	16#432D: sMsg := '432D parameter "Stepper motor stages for one speed stage not allowed" The value for the number of steps for each speed stage in the set value generation is not allowed.';
	16#432E: sMsg := '432E parameter "DWORD for the interpretation of the axis units not allowed" The value that contains the flags for the interpretation of the position and velocity units is not allowed.';
	16#432F: sMsg := '432F parameter "Maximum velocity not allowed" The value for the maximum permitted velocity is not allowed.';
	16#4330: sMsg := '4330 parameter "Motion monitoring window not allowed" The value for the motion monitoring window is not allowed. V';
	16#4331: sMsg := '4331 parameter "PEH time monitoring not allowed" The value for the activation of the PEH time monitoring is not allowed (PEH: positioning end and halt).';
	16#4332: sMsg := '4332 parameter "PEH monitoring time not allowed" The value for the PEH monitoring time (timeout) is not allowed (PEH: positioning end and halt). Default value: 5 s';
	16#4333: sMsg := '4333 parameter "AXISERR_RANGE_DELAYBREAKRELEASE"';
	16#4334: sMsg := '4334 parameter „AXISERR_RANGE_DATAPERSISTENCE”';
	16#433A: sMsg := '433A parameter „AXISERR_RANGE_POSDIFF_FADING_ACCELERATION”';
	16#433B: sMsg := '433B parameter "Fast Axis Stop Signal TYPE NOT allowed" The value FOR the Signal TYPE OF the Fast Axis StoP is NOT allowed [0...5].';
	16#4340: sMsg := '4340 initialization "Axis initialisation" Axis has not been initialised. Although the axis has been created, the rest of the initialisation has not been performed (1. Initialisation of axis I/O, 2. Initialisation of axis…';
	16#4341: sMsg := '4341 address "Group address" Axis does not have a group, or the group address has not been initialised (group contains the set value generation).';
	16#4342: sMsg := '4342 address "Encoder address" The axis does not have an encoder, or the encoder address has not been initialised.';
	16#4343: sMsg := '4343 address "Controller address" The axis does not have a controller, or the controller address has not been initialised.';
	16#4344: sMsg := '4344 address "Drive address" The axis does not have a drive, or the drive address has not been initialised.';
	16#4345: sMsg := '4345 address "Axis interface PLC to NC address" Axis does not have an axis interface from the PLC to the NC, or the axis interface address has not been initialised.';
	16#4346: sMsg := '4346 address "Axis interface NC to PLC address" Axis does not have an axis interface from the NC to the PLC, or the axis interface address has not been initialised.';
	16#4347: sMsg := '4347 address "Size of axis interface NC to PLC is not allowed" (INTERNAL ERROR) The size of the axis interface from NC to PLC is not allowed.';
	16#4348: sMsg := '4348 address "Size of axis interface PLC to NC is not allowed" (INTERNAL ERROR) The size of the axis interface from PLC to NC is not allowed.';
	16#4356: sMsg := '4356 monitoring "Controller enable" Controller enable for the axis is not present (see axis interface SPS®NC). This enable is required, for instance, for an axis positioning task.';
	16#4357: sMsg := '4357 monitoring "Feed enable minus" Feed enable for movement in the negative direction is not present (see axis interface SPS®NC). This enable is required, for instance, for an axis positioning task in the negative d…';
	16#4358: sMsg := '4358 monitoring "Feed enable plus" Feed enable for movement in the positive direction is not present (see axis interface SPS®NC). This enable is required, for instance, for an axis positioning task in the positive di…';
	16#4359: sMsg := '4359 monitoring "Set velocity not allowed" The set velocity requested for a positioning task is not allowed. This can happen if the velocity is less than or equal to zero, larger than the maximum permitted axis veloc…';
	16#435A: sMsg := '435A monitoring "Movement smaller than one encoder increment" (INTERNAL ERROR) The movement required of an axis is, in relation to a positioning task, smaller than one encoder increment (see scaling factor). This inf…';
	16#435B: sMsg := '435B monitoring "Set acceleration monitoring" (INTERNAL ERROR) The set acceleration has exceeded the maximum permitted acceleration or deceleration parameters of the axis.';
	16#435C: sMsg := '435C monitoring "PEH time monitoring" The PEH time monitoring has detected that, after the PEH monitoring time that follows a positioning has elapsed, the target position window has not been reached. The following po…';
	16#435D: sMsg := '435D monitoring "Encoder existence monitoring / movement monitoring" During the active positioning the actual encoder value has changed continuously for a default check time from NC cycle to NC cycle less than the de…';
	16#435E: sMsg := '435E monitoring „Looping distance less than breaking distance” The absolute value of the looping distance is less or equal than the positive or negative breaking distance. This is not allowed.';
	16#4361: sMsg := '4361 monitoring „Time range exceeded (future)” The calculated position lies too far in the future (e.g. when converting a position value in a DC time stamp).';
	16#4362: sMsg := '4362 monitoring „Time range exceeded (past)” The calculated position lies too far in the past (e.g. when converting a position value in a DC time stamp).';
	16#4363: sMsg := '4363 monitoring „Position cannot be determined” The requested position cannot be determined.';
	16#43A0: sMsg := '43A0 internal "Axis consequential error" Consequential error resulting from another causative error related to another axis. Axis consequential errors can occur in relation to master/slave couplings or with multipl…';
	16#4400: sMsg := '4400 parameter "Encoder ID not allowed" The value for the encoder ID is not allowed, e.g. because it has already been assigned, is less than or equal to zero, or is bigger than 255.';
	16#4401: sMsg := '4401 parameter "Encoder type not allowed" The value for the encoder type is unacceptable because it is not defined. Type 1: Simulation (incremental) Type 2: M3000 (24 bit absolute) Type 3: M31x0 (24 bit incremental)…';
	16#4402: sMsg := '4402 parameter "Encoder mode" The value for the encoder (operating) mode is not allowed. Mode 1: Determination of the actual position Mode 2: Determination of the actual position and the actual velocity (filter)';
	16#4403: sMsg := '4403 parameter "Encoder counting direction inverted?" The flag for the encoder counting direction is not allowed. Flag 0: Positive encoder counting direction Flag 1: Negative encoder counting direction';
	16#4404: sMsg := '4404 initialization "Referencing status" The flag for the referencing status is not allowed. Flag 0: Axis has not been referenced Flag 1: Axis has been referenced';
	16#4405: sMsg := '4405 parameter "Encoder increments for each physical encoder rotation" The value for the number of encoder increments for each physical rotation of the encoder is not allowed. This value is used by the software for …';
	16#4406: sMsg := '4406 parameter "Scaling factor" The value for the scaling factor is not allowed. This scaling factor provides the weighting for the conversion of an encoder increment (INC) to a physical unit such as millimeters or …';
	16#4407: sMsg := '4407 parameter "Position offset (zero point offset)" The value for the position offset of the encoder is not allowed. This value is added to the calculated encoder position, and is interpreted in the physical units …';
	16#4408: sMsg := '4408 parameter "Modulo factor" The value for the encoders modulo factor is not allowed.';
	16#4409: sMsg := '4409 parameter "Position filter time" The value for the actual position filter time is not allowed (P-T1 filter).';
	16#440A: sMsg := '440A parameter "Velocity filter time" The value for the actual velocity filter time is not allowed (P-T1 filter).';
	16#440B: sMsg := '440B parameter "Acceleration filter time" The value for the actual acceleration filter time is not allowed (P-T1 filter).';
	16#440C: sMsg := '440C initialization "Cycle time not allowed" (INTERNAL ERROR) The value of the SAF cycle time for the calculation of actual values is not allowed (e.g. is less than or equal to zero).';
	16#440D: sMsg := '440D initialization "" ENCERR_RANGE_UNITFLAGS';
	16#440E: sMsg := '440E parameter "Actual position correction / measurement system error correction" The value for the activation of the actual position correction ("measuring system error correction") is not allowed.';
	16#440F: sMsg := '440F parameter "Filter time actual position correction" The value for the actual position correction filter time is not allowed (P-T1 filter).';
	16#4410: sMsg := '4410 parameter "Search direction for referencing cam inverted" The value of the search direction of the referencing cam in a referencing procedure is not allowed. Value 0: Positive direction Value 1: Negative direct…';
	16#4411: sMsg := '4411 parameter "Search direction for sync pulse (zero pulse) inverted" The value of the search direction of the sync pulse (zero pulse) in a referencing procedure is not allowed. Value 0: Positive direction Value 1:…';
	16#4412: sMsg := '4412 parameter "Reference position" The value of the reference position in a referencing procedure is not allowed.';
	16#4413: sMsg := '4413 parameter "Clearance monitoring between activation of the hardware latch and appearance of the sync pulse" (NOT IMPLEMENTED) The flag for the clearance monitoring between activation of the hardware latch and oc…';
	16#4414: sMsg := '4414 parameter "Minimum clearance between activation of the hardware latch and appearance of the sync pulse" (NOT IMPLEMENTED) The value for the minimum clearance in increments between activation of the hardware lat…';
	16#4415: sMsg := '4415 parameter "External sync pulse" (NOT IMPLEMENTED) The value of the activation or deactivation of the external sync pulse in a referencing procedure is not allowed. Value 0: Passive Value 1: Active';
	16#4416: sMsg := '4416 parameter "Scaling of the noise rate is not allowed" The value of the scaling (weighting) of the synthetic noise rate is not allowed. This parameter exists only in the simulation encoder and serves to produce a…';
	16#4417: sMsg := '4417 parameter „Tolerance window for modulo-start” The value for the tolerance window for the modulo-axis-start is invalid. The value must be greater or equal than zero and smaller than the half encoder modulo-perio…';
	16#4418: sMsg := '4418 parameter „Encoder reference mode” The value for the encoder reference mode is not allowed, resp. is not supported for this encoder type.';
	16#4419: sMsg := '4419 parameter „Encoder evaluation direction” The value for the encoder evaluation direction (log. counter direction) is not allowed.';
	16#441A: sMsg := '441A parameter „Encoder reference system” The value for the encoder reference system is invalid (0: incremental, 1: absolute, 2: absolute+modulo).';
	16#441B: sMsg := '441B parameter „Encoder position initialization mode” When starting the TC system the value for the encoder position initialization mode is invalid.';
	16#441C: sMsg := '441C parameter „Encoder sign interpretation (UNSIGNED- / SIGNED- data type)” The value for the encoder sign interpretation (data type) for the encoder the actual increment calculation (0: Default/not defined, 1: UNS…';
	16#4420: sMsg := '4420 parameter "Software end location monitoring minimum not allowed" The value for the activation of the software location monitoring minimum is not allowed.';
	16#4421: sMsg := '4421 parameter "Software end location monitoring maximum not allowed" The value for the activation of the software location monitoring maximum is not allowed.';
	16#4422: sMsg := '4422 function "Actual value setting is outside the value range" The "set actual value" function cannot be carried out, because the new actual position is outside the expected range of values.';
	16#4423: sMsg := '4423 parameter "Software end location minimum not allowed" The value for the software end location minimum is not allowed.';
	16#4424: sMsg := '4424 parameter "Software end location maximum not allowed" The value for the software end location maximum is not allowed.';
	16#4425: sMsg := '4425 parameter „Filter mask for the raw data of the encoder is invalid” The value for the filter mask of the encoder raw data in increments is invalid.';
	16#4426: sMsg := '4426 parameter „Reference mask for the raw data of the encoder is invalid” The value for the reference mask (increments per encoder turn, absolute resolution) for the raw data of the encoder is invalid. E.g. this va…';
	16#4430: sMsg := '4430 function "Hardware latch activation (encoder)" Activation of the encoder hardware latch was implicitly initiated by the referencing procedure. If this function has already been activated but a latch value has …';
	16#4431: sMsg := '4431 function "External hardware latch activation (encoder)" The activation of the external hardware latch (only available on the KL5101) is initiated explicitly by an ADS command (called from the PLC program of th…';
	16#4432: sMsg := '4432 function "External hardware latch activation (encoder)" If a referencing procedure has previously been initiated and the hardware still signals a valid latch value ("latch valid"), this function must not be ca…';
	16#4433: sMsg := '4433 function "External hardware latch activation (encoder)" If this function has already been initiated and the hardware is still signaling that the external latch value is still valid ("extern latch valid"), a fu…';
	16#4434: sMsg := '4434 monitoring "Encoder function not supported" An encoder function has been activated that is currently not released for use, or which is not even implemented.';
	16#4435: sMsg := '4435 monitoring „Encoder function is already active” An encoder function can not been activated because this functionality is already active.';
	16#4440: sMsg := '4440 initialization "Encoder initialization" Encoder has not been initialized. Although the axis has been created, the rest of the initialization has not been performed (1. Initialization of axis I/O, 2. Initialization o…';
	16#4441: sMsg := '4441 address "Axis address" The encoder does not have an axis, or the axis address has not been initialized.';
	16#4442: sMsg := '4442 address "I/O input structure address" The drive does not have a valid I/O input address in the process image.';
	16#4443: sMsg := '4443 address "I/O output structure address" The encoder does not have a valid I/O output address in the process image.';
	16#4450: sMsg := '4450 monitoring "Encoder counter underflow monitoring" The encoders incremental counter has underflowed.';
	16#4451: sMsg := '4451 monitoring "Encoder counter overflow monitoring" The encoders incremental counter has overflowed.';
	16#4460: sMsg := '4460 monitoring "Software end location minimum (axis start)" With active monitoring of the software end location for a minimum, a start has been made from a position that lies below the software end location minimum.…';
	16#4461: sMsg := '4461 monitoring "Software end location maximum (axis start)" With active monitoring of the software end location for a maximum, a start has been made from a position that lies above the software end location maximum.…';
	16#4462: sMsg := '4462 monitoring "Software end location minimum (positioning process)" With active monitoring of the software end location for a minimum, the actual position has fallen below the software end location minimum. In the …';
	16#4463: sMsg := '4463 monitoring "Software end location maximum (positioning process)" With active monitoring of the software end location for a maximum, the actual position has exceeded the software end location maximum. In the case…';
	16#4464: sMsg := '4464 monitoring „Encoder hardware error” The drive resp. the encoder system reports a hardware error of the encoder. An optimal error code is displayed in the message of the event log.';
	16#4465: sMsg := '4465 monitoring „Position initialization error at system start” At the first initialization of the set position was this for all initialization trials (without over-/under-flow, with underflow and overflow ) out of t…';
	16#4470: sMsg := '4470 monitoring "SSI transformation fault or not finished" The SSI transformation of the FOX 50 module was faulty for some NC-cycles or did not finished respectively.';
	16#44A2: sMsg := '44A2 monitoring "ENCERR_ADDR_CONTROLLER"';
	16#44A3: sMsg := '44A3 monitoring "ENCERR_INVALID_CONTROLLERTYPE"';
	16#4500: sMsg := '4500 parameter "Controller ID not allowed" The value for the controller ID is not allowed, e.g. because it has already been assigned, is less than or equal to zero, or is greater than 255.';
	16#4501: sMsg := '4501 parameter "Controller type not allowed" The value for the controller type is unacceptable because it is not defined. Type 1: P-controller (position) . . . Type 7: High/low speed controller Type 8: Stepper motor…';
	16#4502: sMsg := '4502 parameter "Controller operating mode not allowed" The value for the controller operating mode is not allowed.';
	16#4503: sMsg := '4503 parameter "Weighting of the velocity pre-control not allowed" The value for the percentage weighting of the velocity pre-control is not allowed. The parameter is pre-set to 1.0 (100%) as standard.';
	16#4504: sMsg := '4504 parameter "Following error monitoring (position) not allowed" The value for the activation of the following error monitoring is not allowed.';
	16#4505: sMsg := '4505 parameter "Following error (velocity) not allowed" The value for the activation of the following error monitoring (velocity) is not allowed.';
	16#4506: sMsg := '4506 parameter "Following error window (position) not allowed" The value for the following error window (maximum allowable following error) is not allowed.';
	16#4507: sMsg := '4507 parameter "Following error filter time (position) not allowed" The value for the following error filter time (position) is not allowed.';
	16#4508: sMsg := '4508 parameter "Following error window (velocity) not allowed" The value for the following error window (velocity) is not allowed.';
	16#4509: sMsg := '4509 parameter "Following error filter time (velocity) not allowed" The value for the following error filter time (velocity) is not allowed.';
	16#4510: sMsg := '4510 parameter "Proportional gain Kv or Kp (position controller) not allowed" The value for the proportional gain (Kv factor or Kp factor) is not allowed.';
	16#4511: sMsg := '4511 parameter "Integral-action time Tn (position controller) not allowed" The value for the integral-action time is not allowed (I proportion of the PID T1 controller).';
	16#4512: sMsg := '4512 parameter "Derivative action time Tv (position controller) not allowed" The value for the derivative action time is not allowed (D proportion of the PID T1 controller).';
	16#4513: sMsg := '4513 parameter "Damping time Td (position controller) not allowed" The value for the damping time is not allowed (D proportion of the PID T1 controller). Suggested value: 0.1 * Tv';
	16#4514: sMsg := '4514 function "Activation of the automatic offset compensation not allowed" Activation of the automatic offset compensation is only possible for certain types of controller (with no I component).';
	16#4515: sMsg := '4515 parameter "Additional proportional gain Kv or Kp (position controller) not allowed" The value for the second term of the proportional gain (Kv factor or Kp factor) is not allowed.';
	16#4516: sMsg := '4516 parameter "Reference velocity for additional proportional gain Kv or Kp (position controller) not allowed" The value for the reference velocity percentage data entry, to which the additional proportional gain i…';
	16#4517: sMsg := '4517 parameter "Proportional gain Pa (acceleration proportion) not allowed" The value for the proportional gain (Pa factor) is not allowed.';
	16#4518: sMsg := '4518 parameter "Proportional gain Kv (velocity controller) not allowed" The value for the proportional gain (Kv factor) is not allowed.';
	16#4519: sMsg := '4519 parameter “Reset time Tn (velocity controller) not allowed” The value for the integral-action time is not allowed (I proportion of the PID T1 controller).';
	16#451A: sMsg := '451A address "CONTROLERR_RANGE_ACCJUMPLIMITINGMODE"';
	16#451B: sMsg := '451B address "CONTROLERR_RANGE_ACCJUMPVALUE"';
	16#451C: sMsg := '451C address "CONTROLERR_RANGE_FILTERTIME"';
	16#451D: sMsg := '451D parameter „Dead zone not allowed” The value for the dead zone from the position error or the velocity error (system deviation) is not allowed (only for complex controller with velocity or torque interface).';
	16#4520: sMsg := '4520 parameter ”Rate time Tv (velocity controller) not allowed” The value for the derivative action time is not allowed (D proportion of the PID T1 controller).';
	16#4521: sMsg := '4521 parameter "Damping time Td (velocity controller) not allowed" The value for the damping time is not allowed (D proportion of the PID T1 controller). Suggested value: 0.1 * Tv';
	16#4522: sMsg := '4522 parameter "CONTROLERR_RANGE_IOUTPUTLIMIT"';
	16#4523: sMsg := '4523 parameter "CONTROLERR_RANGE_DOUTPUTLIMIT"';
	16#4524: sMsg := '4524 parameter "CONTROLERR_RANGE_POSIDISABLEWHENMOVING"';
	16#4540: sMsg := '4540 initialization "Controller initialisation" Controller has not been initialised. Although the controller has been created, the rest of the initialisation has not been performed (1. Initialisation of controller, 2. Re…';
	16#4541: sMsg := '4541 address "Axis address" Controller does not know its axis, or the axis address has not been initialised.';
	16#4542: sMsg := '4542 address "Drive address" Controller does not know its drive, or the drive address has not been initialised.';
	16#4550: sMsg := '4550 monitoring "Following error monitoring (position)" With active following error monitoring (position) a following error exceedance has occurred, whose magnitude is greater than the following error window, and who…';
	16#4551: sMsg := '4551 monitoring "Following error monitoring (velocity)" With active following error monitoring (velocity) a velocity following error exceedance has occurred, whose magnitude is greater than the following error window…';
	16#45A0: sMsg := '45A0 monitoring "CONTROLERR_RANGE_AREA_ASIDE"';
	16#45A1: sMsg := '45A1 monitoring "CONTROLERR_RANGE_AREA_BSIDE"';
	16#45A2: sMsg := '45A2 monitoring "CONTROLERR_RANGE_QNENN"';
	16#45A3: sMsg := '45A3 monitoring "CONTROLERR_RANGE_PNENN"';
	16#45A4: sMsg := '45A4 monitoring "CONTROLERR_RANGE_AXISIDPRESP0"';
	16#4600: sMsg := '4600 parameter "Drive ID not allowed" The value for the drive ID is not allowed, e.g. because it has already been assigned, is less than or equal to zero, or is greater than 255.';
	16#4601: sMsg := '4601 parameter "Drive type not allowed" The value for the drive type is unacceptable because it is not defined.';
	16#4602: sMsg := '4602 parameter "Drive operating mode not allowed" The value for the drive operating mode is not allowed. Modus 1: Standard';
	16#4603: sMsg := '4603 parameter "Motor polarity inverted?" The flag for the motor polarity is not allowed. Flag 0: Positive motor polarity Flag 1: Negative motor polarity';
	16#4604: sMsg := '4604 parameter "Drift compensation/velocity offset (DAC offset)" The value for the drift compensation (DAC offset) is not allowed.';
	16#4605: sMsg := '4605 parameter "Reference velocity (velocity pre-control)" The value for the reference velocity (velocity pre-control) is not allowed.';
	16#4606: sMsg := '4606 parameter "Reference output in percent" The value for the reference output in percent is not allowed. The value 1.0 (100 %) usually corresponds to a voltage of 10.0 V.';
	16#4607: sMsg := '4607 parameter "Quadrant compensation factor" The value for the quadrant compensation factor is not allowed.';
	16#4608: sMsg := '4608 parameter "Velocity reference point in percent" The value for the velocity reference point in percent is not allowed. The value 1.0 corresponds to 100 percent.';
	16#4609: sMsg := '4609 parameter "Output reference point in percent" The value for the output reference point in percent is not allowed. The value 1.0 corresponds to 100 percent.';
	16#460A: sMsg := '460A parameter "Minimum or maximum output limit" The values for the minimum and/or maximum output limit is not allowed. This will happen if the range of values is exceeded, the maximum limit is smaller than the mini…';
	16#460B: sMsg := '460B parameter "DRIVEERR_RANGE_MAXINCREMENT"';
	16#460C: sMsg := '460C parameter "DRIVEERR_RANGE_ DRIVECONTROLDWORD"';
	16#460D: sMsg := '460D parameter "DRIVEERR_RANGE_ RESETCYCLECOUNTER"';
	16#460F: sMsg := '460F parameter „Drive torque output scaling is not allowed” The value for the drive torque output scaling (rotary motor) or the force output scaling (linear motor) is not allowed.';
	16#4610: sMsg := '4610 parameter „Drive velocity output scaling is not allowed” The value for the drive velocity output scaling is not allowed.';
	16#4611: sMsg := '4611 parameter "Profi Drive DSC Proportional gain Kpc (position controller) not allowed" The value for the profi drive DSC proportional gain (Kpc factor) is not allowed.';
	16#4612: sMsg := '4612 parameter „Table-ID is invalid” The value for the table-ID is invalid.';
	16#4613: sMsg := '4613 parameter „Table interpolationtype is invalid” The value for the table interpolation-type is invalid.';
	16#4614: sMsg := '4614 parameter „Outputoffset in percent is invalid” The value for the output offset in percent (+/- 1.0) is invalid.';
	16#4615: sMsg := '4615 parameter „Profi Drive DSC scaling factor for calculating Xerr (position controller) is not allowed” The value as profi drive DSC scaling factor for calculating Xerr is invalid.';
	16#4616: sMsg := '4616 parameter „Drive acceleration output scaling is not allowed” The value for the drive acceleration/deceleration output scaling is not allowed.';
	16#4617: sMsg := '4617 parameter „Drive position output scaling is not allowed” The value for the drive position output scaling is not allowed.';
	16#4620: sMsg := '4620 parameter "Bit mask for stepper motor cycle not allowed" A value in the various stepper motor masks for the cycle concerned is not allowed.';
	16#4621: sMsg := '4621 parameter "Bit mask for stepper motor holding current not allowed" The value for the stepper motor holding mask is not allowed.';
	16#4630: sMsg := '4630 monitoring „Overtemperature” The drive resp. terminal detects an overtemperature alarm.';
	16#4631: sMsg := '4631 monitoring „Undervoltage” The drive resp. terminal detects an undervoltage (supply voltage to low).';
	16#4632: sMsg := '4632 monitoring „Wire breakage in phase A” The drive resp. terminal detects a wire breakage in phase A.';
	16#4633: sMsg := '4633 monitoring „Wire breakage in phase B” The drive resp. terminal detects a wire breakage in phase B.';
	16#4634: sMsg := '4634 monitoring „Overcurrent in phase A” The drive resp. terminal detects an overcurrent in phase A.';
	16#4635: sMsg := '4635 monitoring „Overcurrent in Phase B” The drive resp. terminal detects an overcurrent in phase B.';
	16#4636: sMsg := '4636 monitoring „Torque overload (stall situation)” The drive resp. terminal detects a torque overload (stall situation).';
	16#4640: sMsg := '4640 initialization "Drive initialisation" Drive has not been initialised. Although the drive has been created, the rest of the initialisation has not been performed (1. Initialisation of drive I/O, 2. Initialisation of …';
	16#4641: sMsg := '4641 address "Axis address" Drive does not know its axis, or the axis address has not been initialised.';
	16#4642: sMsg := '4642 address "I/O input structure address" The drive does not have a valid I/O input address in the process image.';
	16#4643: sMsg := '4643 address "I/O output structure address" The drive does not have a valid I/O output address in the process image.';
	16#4650: sMsg := '4650 monitoring "Drive not ready for operation" The drive is not ready for operation. The following are possible causes: - the drive is in failure state (hardware fault) - the drive is in the starting-up stage…';
	16#4651: sMsg := '4651 monitoring "Error in cyclic communication with the drive (life counter)"';
	16#4652: sMsg := '4652 monitoring "Not permitted to change the table ID while the axis is enabled"';
	16#4655: sMsg := '4655 monitoring "Invalid IO data for more than n consecutive nc cycles"';
	16#4A00: sMsg := '4A00 parameter "Table ID not allowed" The value for the table ID is not allowed, e.g. because it has already been assigned, is less than or equal to zero, or is greater than 255.';
	16#4A01: sMsg := '4A01 parameter "Table type not allowed" The value for the table type is unacceptable because it is not defined.';
	16#4A02: sMsg := '4A02 parameter "Number of lines in the table not allowed" The value of the number of lines in the table is not allowed, because, for example, it is smaller than two at linear interpolation and smaller than four at s…';
	16#4A03: sMsg := '4A03 parameter "Number of columns in the table is not allowed" The value of the number of columns in the table is not allowed, because, for example, it is less than or equal to zero (depends upon the type of table o…';
	16#4A04: sMsg := '4A04 parameter "Step size (position delta) not allowed" The value for the step size between two lines (position delta) is not allowed, because, for example, it is less than or equal to zero.';
	16#4A05: sMsg := '4A05 parameter "Period not allowed" The value for the period is not allowed, because, for example, it is less than or equal to zero.';
	16#4A06: sMsg := '4A06 parameter "Table is not monotonic" The value for the step size is not allowed, because, for example, it is less than or equal to zero.';
	16#4A07: sMsg := '4A07 initialization „Table sub type is not allowed” The value for the table sub type is not allowed or otherwise the table class (slave type) do not match up to the table main type.';
	16#4A08: sMsg := '4A08 initialization „Table interpolation type is not allowed” The value for the table interpolation type is allowed.';
	16#4A09: sMsg := '4A09 initialization "Incorrect table main type" The table main type is unknown or otherwise the table class (slave type) do not match up to the table main type.';
	16#4A10: sMsg := '4A10 initialization "Table initialisation" Table has not been initialised. Although the table has been created, the rest of the initialisation has not been performed. For instance, the number of lines or columns may be l…';
	16#4A11: sMsg := '4A11 initialization "Not enough memory" Table could not be created, since there is not enough memory.';
	16#4A12: sMsg := '4A12 function "Function not executed, function not available" The function has not been implemented, or cannot be executed, for the present type of table.';
	16#4A13: sMsg := '4A13 function "Line index not allowed" The start line index or the stop line index to be used for read or write access to the table is not allowed. For instance, the line index may be greater than the total number …';
	16#4A14: sMsg := '4A14 function "Column index not allowed" The start column index or the stop column index to be used for read or write access to the table in not allowed. For instance, the column index may be greater than the total…';
	16#4A15: sMsg := '4A15 function "Number of lines not allowed" The number of lines to be read from or written to the table is not allowed. The number of lines must be an integer multiple of the number of elements in a line (n * numbe…';
	16#4A16: sMsg := '4A16 function "Number of columns not allowed" The number of columns to be read from or written to the table is not allowed. The number of columns must be an integer multiple of the number of elements in a column (n…';
	16#4A17: sMsg := '4A17 function "Error in scaling or in range entry" The entries in the table header are inconsistent, e.g. the validity range is empty. If the error is generated during the run time it is a run time error and stops …';
	16#4A18: sMsg := '4A18 function "Multi table slave out of range" The slave master position is outside the table values for the master. The error is a run-time error, and stops the master/slave group.';
	16#4A19: sMsg := '4A19 function "Solo table underflow" The slave master position is outside the table values for the master. The master value of the equidistant table, to be processed linearly, lies under the first table value. The …';
	16#4A1A: sMsg := '4A1A function "Solo table overflow" The slave master position is outside the table values for the master. The master value of the equidistant table, to be processed linearly, lies above the first table value. The e…';
	16#4A1B: sMsg := '4A1B parameter "Incorrect execution mode" The cyclic execution mode can only be "true" or "false".';
	16#4A1C: sMsg := '4A1C parameter "Impermissible parameter" The Fifo parameter is not allowed.';
	16#4A1D: sMsg := '4A1D parameter "Fifo is empty" The Fifo of the external generator is empty. This can signify end of track or a run time error.';
	16#4A1E: sMsg := '4A1E parameter "Fifo is full" The Fifo of the external generator is full. It is the user‘s task to continue to attempt to fill the Fifo with the rejected values.';
	16#4A1F: sMsg := '4A1F parameter „Point-Index of Motion Function invalid” The point index of a Motion Function Point of a Function Table is invalid. First the point index has to be larger than zero and second it has to be numerical c…';
	16#4A20: sMsg := '4A20 initialization „No diagonalisation of matrix” The spline can not be calculated. The master positions are not correct.';
	16#4A21: sMsg := '4A21 initialization „Number of spline points to less” The number of points of a cubic spline has to be greater than two.';
	16#4A22: sMsg := '4A22 initialization „Fifo must not be overwritten” Fifo must not be overwritten since then the active line would be overwritten. It is the task of the user to secure that the active line is not modified.';
	16#4B00: sMsg := '4B00 parameter "Axis has been stopped" The axis has been stopped while the axis moves to target position. The axis could be stopped with a PLC Command via ADS, with the call of AXFNC or with the TwinCAT System Manag…';
	16#4B01: sMsg := '4B01 parameter "Axis cannot be started" The axis cannot be started, because:';
	16#4B02: sMsg := '4B02 parameter "Control mode not allowed" No Target Position Control and no Position Area Control.';
	16#4B03: sMsg := '4B03 parameter "Axis is not moving" Restart position and velocity is only allowed if axis is physically moving.';
	16#4B04: sMsg := '4B04 parameter "Wrong mode for RestartPosAndVelo" Wrong mode.';
	16#4B05: sMsg := '4B05 parameter "Command not allowed"';
	16#4B06: sMsg := '4B06 parameter "Parameter not correct"';
	16#4B07: sMsg := '4B07 parameter "Timeout axis function block"';
	16#4B08: sMsg := '4B08 parameter "Axis in protected mode" Axis is in protected mode (i.e. coupled) and cannot be moved.';
	16#4B09: sMsg := '4B09 parameter "Axis is not ready" Axis is not ready and cannot be moved.';
	16#4B0A: sMsg := '4B0A parameter "Homing error" The Homing of an axis could not be started or was not successful';
	16#4B0B: sMsg := '4B0B parameter "Invalid definition trigger input definition" The definition of the trigger signal used with the function block MC_TouchProbe is invalid. The defined encoder ID, the trigger signal or the trigger sign…';
	16#4B0C: sMsg := '4B0C function "position latch has been deactivated" The function block MC_TouchProbe encountered that a touch probe sequence has been deactivated after the block started this sequence. The reason for instance can b…';
	16#4B0D: sMsg := '4B0D function "Timeout NC status feedback" A function block has successfully executed a command but the NC does not pass the expected feedback in the axis status word.';
	16#4B0E: sMsg := '4B0E function "Supplement not installed" - The function is available as supplement product but not installed on the system.';
	16#4B0F: sMsg := '4B0F function "Timeout Register Access" - The access to a bus terminal register timed out.';
	16#4B10: sMsg := '4B10 function "M-Function request missing" This error occurs if a confirmation of an M-Function is made but the request bit is not set.';
	16#4B11: sMsg := '4B11 parameter "Zero shift index is out of range" The index of the zero shift is invalid';
	16#4B12: sMsg := '4B12 parameter "R parameter index or size is invalid". This error occurs, if the R parameters are written or read and the index or size is out of range';
	16#4B13: sMsg := '4B13 parameter "Index for tool description is invalid"';
	16#4B14: sMsg := '4B14 function "Version of cyclic channel interface does not match to the requested function and function block, resp." This error occurs, if an older TwinCAT Version is used and a new functionality from a newer TcN…';
	16#4B15: sMsg := '4B15 function "Channel is not ready for requested function". The requested function can not be executed due to a wrong state of the channel. This error occurs for instance, if retrace is requested and the axes are …';
	16#4B16: sMsg := '4B16 function "Requested function is not turned on". The requested function requires an explicit activation before it can be executed.';
	16#4B20: sMsg := '4B20 parameter "Cannot append all axes". This error occurs, if you want to append an auxiliary axes to an interpolation group and the function fails. Probably a prior assignment of an auxiliary axes was skipped.';
	16#4B30: sMsg := '4B30 parameter "Pointer invalid". The pointer to a data structure is invalid, e.g. NULL.';
	16#4B31: sMsg := '4B31 parameter "Size of memory invalid". The size parameter is invalid.';
	16#4B32: sMsg := '4B32 parameter "Invalid cam table ID". The cam table ID is out of the range from 1 to 255.';
	16#4B33: sMsg := '4B33 parameter "Invalid point ID". The point ID of a motion function point is lower than 1.';
	16#4B34: sMsg := '4B34 parameter "Invalid number of points ". The number of points to read or write is less than 1.';
	16#4B35: sMsg := '4B35 parameter "Invalid MC table type". The type of a cam table does not match the MC_TableType definition.';
	16#4B36: sMsg := '4B36 parameter "Invalid number of rows". The number of rows of a cam table is less than 1.';
	16#4B37: sMsg := '4B37 parameter "Invalid number of columns". The number of columns of a cam table is invalid.';
	16#4B38: sMsg := '4B38 parameter "Invalid Increment". The increment for an interpolation is invalid, e.g. <= 0.';
	16#4B40: sMsg := '4B40 monitoring "Unsupported Terminal Type". The terminal in use is not supported by this function block.';
	16#4B41: sMsg := '4B41 monitoring "Register Read/Write Error". This error implies to be a validation error.';
	16#4B42: sMsg := '4B42 monitoring "Axis is Enabled". Axis is enabled and is not supposed to be enabled for this operation';
	16#4B43: sMsg := '4B43 parameter "Size of compensation table wrong". The stated table size in bytes is not conform with the real size.';
	16#4B44: sMsg := '4B44 parameter The minimum/ maximum position of the compenstation table is not conform to the position in the table description (ST_CompensationDesc)';
	16#4B45: sMsg := '4B45 parameter "Not implemented". The requested function is not implemented in this combination.';
	16#4B60: sMsg := '4B60 monitoring "Motion command not be activated". A motion command has been started and has been buffered and confirmed by the NC. Nevertheless the command did not become active.';
	16#4B61: sMsg := '4B61 monitoring "Motion command could not be monitored by the PLC". A motion command has been started and has been buffered and confirmed by the NC. The PLC has not been able to monitor the execution of this command……';
	16#4B62: sMsg := '4B62 monitoring "Buffered command finished with error". A buffered command finished with an error. The error number is not available because a new command is already in execution.';
	16#4B63: sMsg := '4B63 monitoring "Buffered command finished without state feedback". A buffered command finished without success or error feedback.';
	16#4B64: sMsg := '4B64 monitoring "  BufferMode  not supported". The  BufferMode  is not supported by the command.';
	16#4B65: sMsg := '4B65 monitoring "Command number is zero". The system administrated command number for buffered commands is zero. ';
	16#4B71: sMsg := '4B71 parameter "Invalid NCI Entry Type". FB_NciFeedTablePreparation is called with an unknown nEntryType';
	16#4B72: sMsg := '4B72 function "NciFeedTable full". The table is full filled and therefore this entry is not accepted.';
	16#4B73: sMsg := '4B73 function internal error';
	16#4B74: sMsg := '4B74 parameter "ST_NciTangentialFollowingDesc: tangential axis is not an auxiliary axis" The entry ST_NciTangentialFollowingDesc contains an tangential axis that is no auxiliary axis.';
	16#4B75: sMsg := '4B75 parameter ST_NciTangentialFollowingDesc: nPathAxis1 and nPathAxis2, resp. are no path axes. So it is not possible to determine the plane.';
	16#4B76: sMsg := '4B76 parameter ST_NciTangentialFollwoingDesc: nPathAxis1 and nPathAxis2 are equal. So it is not possible to determine the plane.';
	16#4B77: sMsg := '4B77 parameter ST_NciGeoCirclePlane: circle is programmed in a wrong manner.';
	16#4B78: sMsg := '4B78 function Internal error in calculation of the tangential following';
	16#4B79: sMsg := '4B79 monitoring Tangential following: With ST_NciTangentialFollowingDesc the monitoring of the deviation angle (E_TfErrorOnCrirical1) is activated and with the actual segment the deviation angle is too big.';
	16#4B7A: sMsg := '4B7A function not implemented';
	16#4B7B: sMsg := '4B7B parameter Tangential Following: The radius of the actual circle segment is too small';
	16#4B7C: sMsg := '4B7C parameter FB_NciFeedTablePreparation: pEntry is NULL';
	16#4B7D: sMsg := '4B7D parameter FB_NciFeedTablePreparation: The specified nEntryType does not match the the structure type';
	16#4B7E: sMsg := '4B7E parameter ST_NciMFuncFast and ST_NciMFuncHsk: The requested m-function is not in between 0..159';
	16#4B7F: sMsg := '4B7F parameter ST_NciDynOvr: The requested value for the dynamic override is not in between 0.01 and 1.0';
	16#4B80: sMsg := '4B80 parameter ST_NciVertexSmoothing: invalid parameter. This error occurs with a negative vertex radius or an unknown vertex smoothing type.';
	16#4B81: sMsg := '4B81 parameter FB_NciFeedTablePrepartion: The requested velocity is not in a valid range';
	16#4B82: sMsg := '4B82 parameter ST_Nci*: invalid parameter';

ELSE
	sMsg := UDINT_TO_STRING(iErrID);
	sMsg := concat(sMsg, ' Unknown Error code');
END_CASE
F_AxErrMsg := sMsg;

END_FUNCTION

// ---- POUs/POUsAxisOnline/AX5000/F_AX5xErrMsg.TcPOU
//==================================================================================================
//							Beckhoff Automation Poland
//								7.12.2018
//		Funkcja konwertujaca nr bledu na opis
// 	v1.0	|| TC v 3.1.4022.27	|| - pierwsza wersja
//==================================================================================================
FUNCTION F_AX5xErrMsg : STRING(255)
VAR_INPUT
	uiDriveError : UINT;
END_VAR

IF uiDriveError < 1 THEN
	F_AX5xErrMsg := '';
	RETURN;
END_IF

CASE uiDriveError OF
	16#1001: F_AX5xErrMsg:= '1001 =  No valid IDN';
	16#1009: F_AX5xErrMsg:= '1009 =  Invalid access to element 1';
	16#2001: F_AX5xErrMsg:= '2001 =  No name';
	16#2002: F_AX5xErrMsg:= '2002 =  Name transmission too short';
	16#2003: F_AX5xErrMsg:= '2003 =  Name transmission too long';
	16#2004: F_AX5xErrMsg:= '2004 =  Name cannot be changed';
	16#2005: F_AX5xErrMsg:= '2005 =  Name is write protected at this time';
	16#3002: F_AX5xErrMsg:= '3002 =  Attribute transmission too short';
	16#3003: F_AX5xErrMsg:= '3003 =  Attribute transmission too long';
	16#3004: F_AX5xErrMsg:= '3004 =  Attribute cannot be changed';
	16#3005: F_AX5xErrMsg:= '3005 =  Attribute is write protected at this time';
	16#4001: F_AX5xErrMsg:= '4001 =  No Unit';
	16#4002: F_AX5xErrMsg:= '4002 =  Unit transmission too short';
	16#4003: F_AX5xErrMsg:= '4003 =  Unit transmission too long';
	16#4004: F_AX5xErrMsg:= '4004 =  Unit cannot be changed';
	16#4005: F_AX5xErrMsg:= '4005 =  Unit is write protected at this time';
	16#5001: F_AX5xErrMsg:= '5001 =  No minimum input value';
	16#5002: F_AX5xErrMsg:= '5002 =  Minimum input value transmission too short';
	16#5003: F_AX5xErrMsg:= '5003 =  Minimum input value transmission too long';
	16#5004: F_AX5xErrMsg:= '5004 =  Minimum input value cannot be changed';
	16#5005: F_AX5xErrMsg:= '5005 =  Minimum input value is write protected at this time';
	16#6001: F_AX5xErrMsg:= '6001 =  No maximum input value';
	16#6002: F_AX5xErrMsg:= '6002 =  Maximum input value transmission too short';
	16#6003: F_AX5xErrMsg:= '6003 =  Maximum input value transmission too long';
	16#6004: F_AX5xErrMsg:= '6004 =  Maximum input value cannot be changed';
	16#6005: F_AX5xErrMsg:= '6005 =  Maximum input value is write protected at this time';
	16#7002: F_AX5xErrMsg:= '7002 =  Operation data value transmission too short';
	16#7003: F_AX5xErrMsg:= '7003 =  Operation data value transmission too long';
	16#7004: F_AX5xErrMsg:= '7004 =  Operation data value cannot be changed';
	16#7005: F_AX5xErrMsg:= '7005 =  Operation data value is write protected at this time';
	16#7006: F_AX5xErrMsg:= '7006 =  Operation data value is smaller than the minimum input value';
	16#7007: F_AX5xErrMsg:= '7007 =  Operation data value is greater than the maximum input value';
	16#7008: F_AX5xErrMsg:= '7008 =  Invalid operation data';
	16#7009: F_AX5xErrMsg:= '7009 =  Operation data is write protected by a password';
	16#7010: F_AX5xErrMsg:= '7010 =  Procedure command already active';
	16#7011: F_AX5xErrMsg:= '7011 =  Procedure command not interruptible';
	16#7012: F_AX5xErrMsg:= '7012 =  Procedure command is at this time not executable';
	16#7013: F_AX5xErrMsg:= '7013 =  Procedure command not executable';
	16#7014: F_AX5xErrMsg:= '7014 =  No data state';
	16#8001: F_AX5xErrMsg:= '8001 =  No default value';
	16#8002: F_AX5xErrMsg:= '8002 =  Default value transmission too long';
	16#8004: F_AX5xErrMsg:= '8004 =  Default value cannot be changed';
	16#700A: F_AX5xErrMsg:= '700A =  Operation data value is write protected';
	16#700B: F_AX5xErrMsg:= '700B =  Invalid indirect addressing';
	16#700C: F_AX5xErrMsg:= '700C =  Operation data is write protected due to other settings';
	16#700D: F_AX5xErrMsg:= '700D =  Reserved';
	16#800A: F_AX5xErrMsg:= '800A =  Invalid drive number';
	16#800B: F_AX5xErrMsg:= '800B =  General error';
	16#800C: F_AX5xErrMsg:= '800C =  No element addressed';
	16#CCD0: F_AX5xErrMsg:= 'CCD0 =  Leaving positive limit switch';
	16#CCD1: F_AX5xErrMsg:= 'CCD1 =  Leaving negative limit switch';
	16#CD40: F_AX5xErrMsg:= 'CD40 =  Clear warning: Overload internal brake resistor';
	16#CD41: F_AX5xErrMsg:= 'CD41 =  Clear warning: Overload external brake resistor';
	16#CD42: F_AX5xErrMsg:= 'CD42 =  Clear warning: Overtemperature amplifier';
	16#CD43: F_AX5xErrMsg:= 'CD43 =  Clear warning: Undervoltage DC link';
	16#CD46: F_AX5xErrMsg:= 'CD46 =  Clear warning: U_mains too high';
	16#CD47: F_AX5xErrMsg:= 'CD47 =  Clear warning: U_mains too low';
	16#D000: F_AX5xErrMsg:= 'D000 =  Esc state: Init';
	16#D001: F_AX5xErrMsg:= 'D001 =  Esc state: PreOp';
	16#D002: F_AX5xErrMsg:= 'D002 =  Esc state: Boot';
	16#D003: F_AX5xErrMsg:= 'D003 =  Esc state: SafeOp';
	16#D005: F_AX5xErrMsg:= 'D005 =  Esc state: Op';
	16#D006: F_AX5xErrMsg:= 'D006 =  Esc state: invalid';
	16#D010: F_AX5xErrMsg:= 'D010 =  Axis state machine: Control section not ready';
	16#D011: F_AX5xErrMsg:= 'D011 =  Axis state machine: Control section ready';
	16#D012: F_AX5xErrMsg:= 'D012 =  Axis state machine: Control and power section ready';
	16#D013: F_AX5xErrMsg:= 'D013 =  Axis state machine: Axis in operation';
	16#D014: F_AX5xErrMsg:= 'D014 =  Axis state machine: Axis halt';
	16#D015: F_AX5xErrMsg:= 'D015 =  Axis state machine: Axis error';
	16#D019: F_AX5xErrMsg:= 'D019 =  Axis state machine: Invalid state';
	16#D101: F_AX5xErrMsg:= 'D101 =  Hardware enable not active.';
	16#D102: F_AX5xErrMsg:= 'D102 =  Safety card active,  AX5000 in the safe condition';
	16#D180: F_AX5xErrMsg:= 'D180 =  SCI communication Control - Front pcb: Frame error';
	16#D181: F_AX5xErrMsg:= 'D181 =  SCI communication Control - Front pcb: Parity error';
	16#D182: F_AX5xErrMsg:= 'D182 =  SCI communication Control - Front pcb: RX-Data missing';
	16#D183: F_AX5xErrMsg:= 'D183 =  SCI communication Control - Front pcb: SCI error';
	16#D184: F_AX5xErrMsg:= 'D184 =  SCI communication Control - Front pcb: Timeout error';
	16#D185: F_AX5xErrMsg:= 'D185 =  SCI communication Control - Front pcb: Checksum error';
	16#D186: F_AX5xErrMsg:= 'D186 =  SCI communication Control - Front pcb: Byte count error';
	16#D187: F_AX5xErrMsg:= 'D187 =  SCI communication Control - Front pcb: Command denied';
	16#D188: F_AX5xErrMsg:= 'D188 =  SCI communication Control - Front pcb: Wrong command';
	16#D189: F_AX5xErrMsg:= 'D189 =  SCI communication Control - Front pcb: Command error';
	16#D18A: F_AX5xErrMsg:= 'D18A =  SCI communication Control - Front pcb: Timeout error';
	16#D18B: F_AX5xErrMsg:= 'D18B =  SCI communication Control - Front pcb: RX data error';
	16#D18C: F_AX5xErrMsg:= 'D18C =  SCI communication Control - Front pcb: Wrong channel';
	16#D18D: F_AX5xErrMsg:= 'D18D =  SCI communication Control - Front pcb: Fifo overflow';
	16#D18E: F_AX5xErrMsg:= 'D18E =  SCI communication Front - Control pcb: Frame error';
	16#D18F: F_AX5xErrMsg:= 'D18F =  SCI communication Front - Control pcb: Parity error';
	16#D190: F_AX5xErrMsg:= 'D190 =  SCI communication Front - Control pcb: Wrong checksum';
	16#D191: F_AX5xErrMsg:= 'D191 =  SCI communication Front - Control pcb: Timeout error';
	16#D192: F_AX5xErrMsg:= 'D192 =  SCI communication Front - Control pcb: Response timeout error';
	16#D193: F_AX5xErrMsg:= 'D193 =  SCI communication Front - Control pcb: Fifo overflow';
	16#D194: F_AX5xErrMsg:= 'D194 =  SCI communication Control - Front pcb: SCI reset called';
	16#D195: F_AX5xErrMsg:= 'D195 =  SCI communication Control - Front pcb: Byte count error';
	16#D196: F_AX5xErrMsg:= 'D196 =  SCI communication Control - Front pcb: Buffer overflow';
	16#D1B0: F_AX5xErrMsg:= 'D1B0 =  SCI communication Control - Option card: Frame error';
	16#D1B1: F_AX5xErrMsg:= 'D1B1 =  SCI communication Control - Option card: Parity error';
	16#D1B2: F_AX5xErrMsg:= 'D1B2 =  SCI communication Control - Option card: RX-Data missing';
	16#D1B3: F_AX5xErrMsg:= 'D1B3 =  SCI communication Control - Option card: SCI error';
	16#D1B4: F_AX5xErrMsg:= 'D1B4 =  SCI communication Control - Option card: Timeout error';
	16#D1B5: F_AX5xErrMsg:= 'D1B5 =  SCI communication Control - Option card: Checksum error';
	16#D1B6: F_AX5xErrMsg:= 'D1B6 =  SCI communication Control - Option card: Byte count error';
	16#D1B7: F_AX5xErrMsg:= 'D1B7 =  SCI communication Control - Option card: Command denied';
	16#D1B8: F_AX5xErrMsg:= 'D1B8 =  SCI communication Control - Option card: Wrong command';
	16#D1B9: F_AX5xErrMsg:= 'D1B9 =  SCI communication Control - Option card: Command error';
	16#D1BA: F_AX5xErrMsg:= 'D1BA =  SCI communication Control - Option card: Timeout error';
	16#D1BB: F_AX5xErrMsg:= 'D1BB =  SCI communication Control - Option card: RX data error';
	16#D1BC: F_AX5xErrMsg:= 'D1BC =  SCI communication Control - Option card: Wrong channel';
	16#D1BD: F_AX5xErrMsg:= 'D1BD =  SCI communication Control - Option card: Fifo overflow';
	16#D1BE: F_AX5xErrMsg:= 'D1BE =  SCI communication Front - Control pcb: Frame error';
	16#D1BF: F_AX5xErrMsg:= 'D1BF =  SCI communication Front - Control pcb: Parity error';
	16#D1C0: F_AX5xErrMsg:= 'D1C0 =  SCI communication Front - Control pcb: Wrong checksum';
	16#D1C1: F_AX5xErrMsg:= 'D1C1 =  SCI communication Front - Control pcb: Timeout error';
	16#D1C2: F_AX5xErrMsg:= 'D1C2 =  SCI communication Front - Control pcb: Response timeout error';
	16#D1C3: F_AX5xErrMsg:= 'D1C3 =  SCI communication Front - Control pcb: Fifo overflow';
	16#D1C4: F_AX5xErrMsg:= 'D1C4 =  SCI communication Control - Option card: SCI reset called';
	16#D1C5: F_AX5xErrMsg:= 'D1C5 =  SCI communication Control - Option card: Byte count error';
	16#D1C6: F_AX5xErrMsg:= 'D1C6 =  SCI communication Control - Option card: Buffer overflow';
	16#D200: F_AX5xErrMsg:= 'D200 =  Firmware update successful!';
	16#D400: F_AX5xErrMsg:= 'D400 =  ESC: PLL timeout';
	16#D401: F_AX5xErrMsg:= 'D401 =  ESC: Io-Sync timeout';
	16#D402: F_AX5xErrMsg:= 'D402 =  Info procedure command: state change';
	16#D403: F_AX5xErrMsg:= 'D403 =  Esc state machine: State change active';
	16#D404: F_AX5xErrMsg:= 'D404 =  Esc state machine: Error flag not cleared';
	16#D500: F_AX5xErrMsg:= 'D500 =  External ADC: Uref invalid';
	16#D780: F_AX5xErrMsg:= 'D780 =  Feedback Parameter Channel Endat: Crc Error';
	16#D781: F_AX5xErrMsg:= 'D781 =  Feedback Parameter Channel Endat: Mode crc error';
	16#D782: F_AX5xErrMsg:= 'D782 =  Feedback Parameter Channel Endat: Timeout encoder response';
	16#D783: F_AX5xErrMsg:= 'D783 =  Feedback Parameter Channel Endat: Timeout encoder response';
	16#D784: F_AX5xErrMsg:= 'D784 =  Feedback Parameter Channel Endat: Wrong response';
	16#D786: F_AX5xErrMsg:= 'D786 =  Feedback Parameter Channel Endat: Encoder not ready';
	16#D787: F_AX5xErrMsg:= 'D787 =  Feedback Parameter Channel Endat: Formatting OEM memory';
	16#D808: F_AX5xErrMsg:= 'D808 =  Feedback Parameter Channel Hiperface: Wrong analog channel';
	16#DC30: F_AX5xErrMsg:= 'DC30 =  I2C communication: Save error ID 1';
	16#DC31: F_AX5xErrMsg:= 'DC31 =  I2C communication: Save error ID 2';
	16#DC32: F_AX5xErrMsg:= 'DC32 =  I2C communication: Save parameter';
	16#DC33: F_AX5xErrMsg:= 'DC33 =  I2C communication: Save operation time 1';
	16#DC34: F_AX5xErrMsg:= 'DC34 =  I2C communication: Save operation time 2';
	16#DC35: F_AX5xErrMsg:= 'DC35 =  I2C communication: Read';
	16#DC36: F_AX5xErrMsg:= 'DC36 =  I2C communication: Read';
	16#DC37: F_AX5xErrMsg:= 'DC37 =  I2C communication: Read';
	16#DC38: F_AX5xErrMsg:= 'DC38 =  I2C communication: Write';
	16#DC39: F_AX5xErrMsg:= 'DC39 =  I2C communication: Write';
	16#DC3A: F_AX5xErrMsg:= 'DC3A =  I2C communication: Different operation time';
	16#DC3B: F_AX5xErrMsg:= 'DC3B =  I2C communication: Job buffer full';
	16#DC3C: F_AX5xErrMsg:= 'DC3C =  I2C communication: No safety hardware';
	16#DC3D: F_AX5xErrMsg:= 'DC3D =  I2C communication: No option hardware';
	16#DC3E: F_AX5xErrMsg:= 'DC3E =  I2C communication: Device operation time overflow';
	16#DC3F: F_AX5xErrMsg:= 'DC3F =  I2C communication: Channel operation time overflow';
	16#DCB0: F_AX5xErrMsg:= 'DCB0 =  Lcd: Wrong Esc state';
	16#DCB1: F_AX5xErrMsg:= 'DCB1 =  Lcd: Wrong axis state';
	16#DCB2: F_AX5xErrMsg:= 'DCB2 =  Lcd: Unknown cyclic job';
	16#DCB3: F_AX5xErrMsg:= 'DCB3 =  Lcd: Unknown job';
	16#DCB4: F_AX5xErrMsg:= 'DCB4 =  Lcd: Unknown state';
	16#DCB5: F_AX5xErrMsg:= 'DCB5 =  Lcd: Unknown state';
	16#DCB6: F_AX5xErrMsg:= 'DCB6 =  Lcd: Unknown state';
	16#DCB7: F_AX5xErrMsg:= 'DCB7 =  Lcd: Unknown state';
	16#DCB8: F_AX5xErrMsg:= 'DCB8 =  Lcd: Unknown menue state';
	16#DCB9: F_AX5xErrMsg:= 'DCB9 =  Lcd: Interface error';
	16#DCBA: F_AX5xErrMsg:= 'DCBA =  Lcd: Invalid state';
	16#DCBB: F_AX5xErrMsg:= 'DCBB =  Lcd: Communication error';
	16#DD42: F_AX5xErrMsg:= 'DD42 =  Power management: DC link current in limit';
	16#DD80: F_AX5xErrMsg:= 'DD80 =  Control pcb: Main loop time exceeded';
	16#DD81: F_AX5xErrMsg:= 'DD81 =  Control pcb: End of stack reached';
	16#DD82: F_AX5xErrMsg:= 'DD82 =  Front pcb: Main loop time exceeded';
	16#DD83: F_AX5xErrMsg:= 'DD83 =  Front pcb: End of stack reached';
	16#DFFF: F_AX5xErrMsg:= 'DFFF =  Debug firmware,  replace "As soon as possible"!';
	16#E160: F_AX5xErrMsg:= 'E160 =  Process data mapping: Mapping code of IDN %s could not be copied.';
	16#E290: F_AX5xErrMsg:= 'E290 =  High-priority processes cannot be processed';
	16#E300: F_AX5xErrMsg:= 'E300 =  The IO-Watchdog has been disabled!!!! (User mode debugging!)';
	16#E581: F_AX5xErrMsg:= 'E581 =  External Periphery - Control card: Reading the ESC-eeprom failed';
	16#ECD0: F_AX5xErrMsg:= 'ECD0 =  Positive limit switch warning.';
	16#ECD1: F_AX5xErrMsg:= 'ECD1 =  Negative limit switch warning.';
	16#ED00: F_AX5xErrMsg:= 'ED00 =  Motor overtemperature';
	16#ED01: F_AX5xErrMsg:= 'ED01 =  Overload - motor';
	16#ED40: F_AX5xErrMsg:= 'ED40 =  Overload - Internal brake resistor';
	16#ED41: F_AX5xErrMsg:= 'ED41 =  Overload - External brake resistor';
	16#ED42: F_AX5xErrMsg:= 'ED42 =  Overtemperature - Amplifier';
	16#ED43: F_AX5xErrMsg:= 'ED43 =  Undervoltage - DC link';
	16#ED46: F_AX5xErrMsg:= 'ED46 =  U_mains too high';
	16#ED47: F_AX5xErrMsg:= 'ED47 =  U_mains too low';
	16#ED60: F_AX5xErrMsg:= 'ED60 =  Feedback - Warning bit set';
	16#F010: F_AX5xErrMsg:= 'F010 =  Firmware-Download: Flash error';
	16#F011: F_AX5xErrMsg:= 'F011 =  Firmware-Download: Flash error';
	16#F012: F_AX5xErrMsg:= 'F012 =  Firmware-Download: Flash error';
	16#F013: F_AX5xErrMsg:= 'F013 =  Firmware-Download: Flash error';
	16#F014: F_AX5xErrMsg:= 'F014 =  Firmware-Download: Flash error';
	16#F015: F_AX5xErrMsg:= 'F015 =  Firmware-Download: Flash error';
	16#F016: F_AX5xErrMsg:= 'F016 =  Firmware-Download: Flash error';
	16#F017: F_AX5xErrMsg:= 'F017 =  Firmware-Download: Flash error';
	16#F018: F_AX5xErrMsg:= 'F018 =  Firmware-Download: Flash error';
	16#F019: F_AX5xErrMsg:= 'F019 =  Firmware-Download: Flash error';
	16#F01A: F_AX5xErrMsg:= 'F01A =  Firmware-Download: Flash error';
	16#F01B: F_AX5xErrMsg:= 'F01B =  Firmware-Download: Flash error';
	16#F01C: F_AX5xErrMsg:= 'F01C =  Firmware-Download: Flash error';
	16#F01D: F_AX5xErrMsg:= 'F01D =  Firmware-Download: Flash error';
	16#F01E: F_AX5xErrMsg:= 'F01E =  Firmware-Download: Flash error';
	16#F030: F_AX5xErrMsg:= 'F030 =  Firmware-Download: Invalid file name';
	16#F032: F_AX5xErrMsg:= 'F032 =  Firmware download: Firmware file does not match the device';
	16#F033: F_AX5xErrMsg:= 'F033 =  Firmware-Download: Firmware-File is defective';
	16#F040: F_AX5xErrMsg:= 'F040 =  Firmware-Download: Firmware-File is defective';
	16#F041: F_AX5xErrMsg:= 'F041 =  Firmware-Download: Firmware-File is defective';
	16#F042: F_AX5xErrMsg:= 'F042 =  Firmware-Download: Firmware-File is defective';
	16#F043: F_AX5xErrMsg:= 'F043 =  Firmware-Download: Read of the hardware ID"s failed.';
	16#F044: F_AX5xErrMsg:= 'F044 =  Firmware-Download: Firmware-File is wrong or defective';
	16#F045: F_AX5xErrMsg:= 'F045 =  Firmware-Download: Firmware-File is defective';
	16#F046: F_AX5xErrMsg:= 'F046 =  Firmware-Download: Firmware-File is defective';
	16#F047: F_AX5xErrMsg:= 'F047 =  Firmware-Download: Firmware-File is defective';
	16#F048: F_AX5xErrMsg:= 'F048 =  Firmware-Download: Hardware is defective';
	16#F049: F_AX5xErrMsg:= 'F049 =  Firmware-Download: Hardware is defective';
	16#F04A: F_AX5xErrMsg:= 'F04A =  Firmware-Download: Hardware is defective';
	16#F04B: F_AX5xErrMsg:= 'F04B =  Firmware-Download: Firmware-File is defective';
	16#F04C: F_AX5xErrMsg:= 'F04C =  Firmware-Download: Firmware-File is defective';
	16#F04D: F_AX5xErrMsg:= 'F04D =  Firmware-Download: Firmware-File is defective';
	16#F04E: F_AX5xErrMsg:= 'F04E =  Firmware-Download: Firmware-File is defective';
	16#F04F: F_AX5xErrMsg:= 'F04F =  Firmware-Download: Wrong TwinCAT version';
	16#F050: F_AX5xErrMsg:= 'F050 =  Firmware-Download: Firmware-File is defective';
	16#F051: F_AX5xErrMsg:= 'F051 =  Firmware-Download: Firmware-File is defective';
	16#F052: F_AX5xErrMsg:= 'F052 =  Firmware-Download: Firmware-File is defective';
	16#F053: F_AX5xErrMsg:= 'F053 =  Firmware-Download: Firmware-File is defective';
	16#F054: F_AX5xErrMsg:= 'F054 =  Firmware-Download: Firmware-File is defective';
	16#F055: F_AX5xErrMsg:= 'F055 =  Firmware-Download: Firmware-File is defective';
	16#F056: F_AX5xErrMsg:= 'F056 =  Firmware-Download: Firmware-File is wrong or defective';
	16#F057: F_AX5xErrMsg:= 'F057 =  Firmware-Download: Firmware-File is defective';
	16#F058: F_AX5xErrMsg:= 'F058 =  Firmware-Download: Firmware-File is defective';
	16#F059: F_AX5xErrMsg:= 'F059 =  Firmware-Download: Firmware-File is defective';
	16#F060: F_AX5xErrMsg:= 'F060 =  Firmware-Download: Firmware-File is defective';
	16#F061: F_AX5xErrMsg:= 'F061 =  Firmware-Download: Hardware is defective';
	16#F062: F_AX5xErrMsg:= 'F062 =  Firmware-Download: Hardware is defective';
	16#F063: F_AX5xErrMsg:= 'F063 =  Firmware-Download: Firmware-File or device is defective';
	16#F064: F_AX5xErrMsg:= 'F064 =  Firmware-Download: Firmware-File or device is defective';
	16#F065: F_AX5xErrMsg:= 'F065 =  Firmware-Download: Firmware-File is wrong';
	16#F066: F_AX5xErrMsg:= 'F066 =  Firmware-Download: Firmware-File or device is defective';
	16#F067: F_AX5xErrMsg:= 'F067 =  Firmware-Download: Internal config error';
	16#F068: F_AX5xErrMsg:= 'F068 =  Firmware-Download: Bootloader update required.';
	16#F06A: F_AX5xErrMsg:= 'F06A =  Firmware-Download: Ctrl pcb eeprom not accessible.';
	16#F06B: F_AX5xErrMsg:= 'F06B =  Firmware-Download: Front pcb eeprom not accessible.';
	16#F06C: F_AX5xErrMsg:= 'F06C =  Firmware-Download: Driver pcb eeprom not accessible.';
	16#F06D: F_AX5xErrMsg:= 'F06D =  Firmware-Download: Power pcb eeprom not accessible.';
	16#F06E: F_AX5xErrMsg:= 'F06E =  Firmware-Download: Safety pcb eeprom not accessible.';
	16#F06F: F_AX5xErrMsg:= 'F06F =  Firmware-Download: Safety pcb eeprom not accessible.';
	16#F070: F_AX5xErrMsg:= 'F070 =  Firmware-Download: Firmware index for the control pcb don"t match';
	16#F071: F_AX5xErrMsg:= 'F071 =  Firmware-Download: Firmware index for the front pcb don"t match';
	16#F072: F_AX5xErrMsg:= 'F072 =  Firmware-Download: Firmware index for the driver pcb don"t match';
	16#F073: F_AX5xErrMsg:= 'F073 =  Firmware-Download: Firmware index for the power pcb don"t match';
	16#F074: F_AX5xErrMsg:= 'F074 =  Firmware-Download: Firmware index for the Safety pcb don"t match';
	16#F075: F_AX5xErrMsg:= 'F075 =  Firmware-Download: Firmware index for the option pcb don"t match';
	16#F076: F_AX5xErrMsg:= 'F076 =  Firmware-Download: Firmware index for the control pcb can"t be read';
	16#F077: F_AX5xErrMsg:= 'F077 =  Firmware-Download: Firmware index for the front pcb can"t be read';
	16#F078: F_AX5xErrMsg:= 'F078 =  Firmware-Download: Firmware index for the driver pcb can"t be read';
	16#F079: F_AX5xErrMsg:= 'F079 =  Firmware-Download: Firmware index for the power pcb can"t be read';
	16#F07A: F_AX5xErrMsg:= 'F07A =  Firmware-Download: Firmware index for the safety pcb can"t be read';
	16#F07B: F_AX5xErrMsg:= 'F07B =  Firmware-Download: Firmware index for the option pcb can"t be read';
	16#F090: F_AX5xErrMsg:= 'F090 =  Firmware-Download: FPGA error option pcb';
	16#F091: F_AX5xErrMsg:= 'F091 =  Firmware-Download: FPGA error option pcb';
	16#F092: F_AX5xErrMsg:= 'F092 =  Firmware-Download: FPGA error option pcb';
	16#F093: F_AX5xErrMsg:= 'F093 =  Firmware-Download: FPGA error option pcb';
	16#F094: F_AX5xErrMsg:= 'F094 =  Firmware-Download: FPGA error option pcb';
	16#F095: F_AX5xErrMsg:= 'F095 =  Firmware-Download: FPGA error option pcb';
	16#F096: F_AX5xErrMsg:= 'F096 =  Firmware-Download: FPGA error option pcb';
	16#F0A0: F_AX5xErrMsg:= 'F0A0 =  FPGA error: configuration could not be loaded';
	16#F0A1: F_AX5xErrMsg:= 'F0A1 =  FPGA error: Configuration file is missing';
	16#F0A2: F_AX5xErrMsg:= 'F0A2 =  FPGA error: Loading of the configuration failed.';
	16#F0B0: F_AX5xErrMsg:= 'F0B0 =  Serial Flash error';
	16#F0B1: F_AX5xErrMsg:= 'F0B1 =  Serial Flash error';
	16#F0B2: F_AX5xErrMsg:= 'F0B2 =  Serial Flash error';
	16#F0B3: F_AX5xErrMsg:= 'F0B3 =  Serial Flash error';
	16#F0B4: F_AX5xErrMsg:= 'F0B4 =  Serial Flash error';
	16#F0B5: F_AX5xErrMsg:= 'F0B5 =  Serial Flash error';
	16#F0B6: F_AX5xErrMsg:= 'F0B6 =  Serial Flash error';
	16#F0B7: F_AX5xErrMsg:= 'F0B7 =  Serial Flash error';
	16#F0B8: F_AX5xErrMsg:= 'F0B8 =  Serial Flash error';
	16#F0B9: F_AX5xErrMsg:= 'F0B9 =  Serial Flash error: Bootloader defective';
	16#F0BA: F_AX5xErrMsg:= 'F0BA =  Serial Flash error: Internal firmware file is defective';
	16#F0BB: F_AX5xErrMsg:= 'F0BB =  Serial Flash error: Internal system data file not found';
	16#F0BC: F_AX5xErrMsg:= 'F0BC =  Serial Flash error: Internal system data file is defective';
	16#F0BD: F_AX5xErrMsg:= 'F0BD =  Serial Flash error: Initialization failed';
	16#F0BE: F_AX5xErrMsg:= 'F0BE =  Serial Flash error: Processing failed';
	16#F0BF: F_AX5xErrMsg:= 'F0BF =  Serial Flash error: Write error';
	16#F0C0: F_AX5xErrMsg:= 'F0C0 =  Serial Flash error: Diagnostics file not found';
	16#F0C1: F_AX5xErrMsg:= 'F0C1 =  Serial Flash error: Internal error';
	16#F100: F_AX5xErrMsg:= 'F100 =  Axis state machine: Communication error';
	16#F101: F_AX5xErrMsg:= 'F101 =  Axis state machine: Initialize error';
	16#F102: F_AX5xErrMsg:= 'F102 =  Axis state machine: Loss of the hardware enable';
	16#F103: F_AX5xErrMsg:= 'F103 =  Axis state machine: Got no timer';
	16#F104: F_AX5xErrMsg:= 'F104 =  Axis state machine: NC errorhandling - Timeout';
	16#F105: F_AX5xErrMsg:= 'F105 =  Axis state machine: Maximum drive off delay time elapsed';
	16#F106: F_AX5xErrMsg:= 'F106 =  Axis state machine: No motor configured';
	16#F107: F_AX5xErrMsg:= 'F107 =  Axis state machine: Current control not ready to enable';
	16#F108: F_AX5xErrMsg:= 'F108 =  Axis state machine: Velocity control not ready';
	16#F109: F_AX5xErrMsg:= 'F109 =  Axis state machine: Position control not ready';
	16#F10A: F_AX5xErrMsg:= 'F10A =  Axis state machine: Wake and Shake not idle';
	16#F10B: F_AX5xErrMsg:= 'F10B =  Axis State Machine: Wake and Shake command failed';
	16#F10C: F_AX5xErrMsg:= 'F10C =  Axis State Machine: Not possible to enable';
	16#F10D: F_AX5xErrMsg:= 'F10D =  Axis State Machine: Not possible to enable';
	16#F10E: F_AX5xErrMsg:= 'F10E =  Axis State Machine: The motor connection check failed.';
	16#F10F: F_AX5xErrMsg:= 'F10F =  Axis State Machine: The configured error propagation input isn"t active.';
	16#F120: F_AX5xErrMsg:= 'F120 =  Command "Motor and feedback check": Timeout';
	16#F121: F_AX5xErrMsg:= 'F121 =  Command "Motor and feedback check": No hardware enable';
	16#F122: F_AX5xErrMsg:= 'F122 =  Command "Motor and feedback connection check"';
	16#F123: F_AX5xErrMsg:= 'F123 =  Command "Motor and feedback check" failed';
	16#F124: F_AX5xErrMsg:= 'F124 =  Reset-Command: Got no timer';
	16#F125: F_AX5xErrMsg:= 'F125 =  Reset-Command: Got no timer';
	16#F126: F_AX5xErrMsg:= 'F126 =  Reset-Command: Initialization failed';
	16#F127: F_AX5xErrMsg:= 'F127 =  Reset-Command: Feedback DSP - timeout';
	16#F128: F_AX5xErrMsg:= 'F128 =  Reset-Command: One or more of the pending errors is not resettable';
	16#F129: F_AX5xErrMsg:= 'F129 =  Reset-Command: Reset is not executable';
	16#F12A: F_AX5xErrMsg:= 'F12A =  Error reaction "Torque off" forced';
	16#F12B: F_AX5xErrMsg:= 'F12B =  Error reaction "Shorted coils brake" forced';
	16#F12C: F_AX5xErrMsg:= 'F12C =  Error reaction "Open loop ramp" forced';
	16#F12D: F_AX5xErrMsg:= 'F12D =  Error reaction "Closed loop ramp" forced';
	16#F12E: F_AX5xErrMsg:= 'F12E =  Error reaction "NC-Handling" forced';
	16#F12F: F_AX5xErrMsg:= 'F12F =  Command "Motor and feedback connection check": No enable permission from the Safety option';
	16#F130: F_AX5xErrMsg:= 'F130 =  Command "Wake and Shake": Timeout';
	16#F131: F_AX5xErrMsg:= 'F131 =  Command "Reset": Feedback initialization failed';
	16#F132: F_AX5xErrMsg:= 'F132 =  Command "Reset": Not possible - Internal hardware error';
	16#F133: F_AX5xErrMsg:= 'F133 =  Command "Reset": Not possible - Drive is still enabled';
	16#F134: F_AX5xErrMsg:= 'F134 =  Command "Reset": Restart of the modulo calculation failed.';
	16#F135: F_AX5xErrMsg:= 'F135 =  Parameterset-Switching: Reactivation of the parameterset 0 failed.';
	16#F136: F_AX5xErrMsg:= 'F136 =  Parameterset-Switching: Switching to parameterset x failed.';
	16#F137: F_AX5xErrMsg:= 'F137 =  Parameterset-Switching: Feature not available';
	16#F138: F_AX5xErrMsg:= 'F138 =  Parameterset-Switching: Axis is in operation,  switching not possible. ';
	16#F139: F_AX5xErrMsg:= 'F139 =  Parameterset-Switching: Internal error.';
	16#F13A: F_AX5xErrMsg:= 'F13A =  Parameterset-Switching: Switching to parameterset x not possible.';
	16#F13B: F_AX5xErrMsg:= 'F13B =  Option card and OCT interface: Reset failed.';
	16#F13C: F_AX5xErrMsg:= 'F13C =  Reset command - Timeout';
	16#F13E: F_AX5xErrMsg:= 'F13E =  error reaction ôFeedback errorö forced';
	16#F13F: F_AX5xErrMsg:= 'F13F =  Creation of the position interpolator failed';
	16#F140: F_AX5xErrMsg:= 'F140 =  Build drive system: Failed';
	16#F141: F_AX5xErrMsg:= 'F141 =  Build drive system: Timeout';
	16#F142: F_AX5xErrMsg:= 'F142 =  Initialization of the current controller failed';
	16#F143: F_AX5xErrMsg:= 'F143 =  Initialization of the velocity controller failed';
	16#F144: F_AX5xErrMsg:= 'F144 =  Initialization of the position controller failed';
	16#F145: F_AX5xErrMsg:= 'F145 =  Initialization of the feedback failed';
	16#F146: F_AX5xErrMsg:= 'F146 =  Build drive system: Failed';
	16#F147: F_AX5xErrMsg:= 'F147 =  Build drive system: Memory error Front card';
	16#F148: F_AX5xErrMsg:= 'F148 =  Build drive system: Unknown feedback system';
	16#F149: F_AX5xErrMsg:= 'F149 =  Build drive system: Front card - Internal error';
	16#F14A: F_AX5xErrMsg:= 'F14A =  Build drive system: Front card û software error';
	16#F14B: F_AX5xErrMsg:= 'F14B =  Build drive system: Memory error Control card';
	16#F14C: F_AX5xErrMsg:= 'F14C =  Build drive system: Memory error Front card';
	16#F14D: F_AX5xErrMsg:= 'F14D =  System memory deallocation: Feedback termination failed';
	16#F14E: F_AX5xErrMsg:= 'F14E =  System memory deallocation: Command error';
	16#F14F: F_AX5xErrMsg:= 'F14F =  System memory deallocation: Command error';
	16#F150: F_AX5xErrMsg:= 'F150 =  Initialization of the feedback: Internal error';
	16#F151: F_AX5xErrMsg:= 'F151 =  Initialization of the feedback: Timeout';
	16#F152: F_AX5xErrMsg:= 'F152 =  Initialisation of the feedback: Command failed';
	16#F153: F_AX5xErrMsg:= 'F153 =  Initialization of the feedback: No option card found';
	16#F154: F_AX5xErrMsg:= 'F154 =  Build drive system: Memory error option card';
	16#F155: F_AX5xErrMsg:= 'F155 =  Build drive system: Option card - Unknown feedback system';
	16#F156: F_AX5xErrMsg:= 'F156 =  Build drive system: Option card - Internal error';
	16#F157: F_AX5xErrMsg:= 'F157 =  Build drive system: Option card - Unknown feedback system';
	16#F158: F_AX5xErrMsg:= 'F158 =  System memory deallocation: Front card - Internal error';
	16#F159: F_AX5xErrMsg:= 'F159 =  System memory deallocation: Option card - Internal error';
	16#F15A: F_AX5xErrMsg:= 'F15A =  Feedback error: Plug connector combination invalid';
	16#F15B: F_AX5xErrMsg:= 'F15B =  Feedback error: No OCT support.';
	16#F15F: F_AX5xErrMsg:= 'F15F =  No control loops allocated. Calibration mode active.';
	16#F160: F_AX5xErrMsg:= 'F160 =  Process data mapping: Internal error';
	16#F161: F_AX5xErrMsg:= 'F161 =  Process data mapping: AT - S-0-0016';
	16#F162: F_AX5xErrMsg:= 'F162 =  Process data mapping: AT - S-0-0016';
	16#F163: F_AX5xErrMsg:= 'F163 =  Process data mapping: AT - Memory problem';
	16#F164: F_AX5xErrMsg:= 'F164 =  Process data mapping: Internal error';
	16#F165: F_AX5xErrMsg:= 'F165 =  Process data mapping: AT - Anzahl der IDN"s';
	16#F166: F_AX5xErrMsg:= 'F166 =  Process data mapping: MDT - S-0-0024';
	16#F167: F_AX5xErrMsg:= 'F167 =  Process data mapping: MDT - S-0-0024';
	16#F168: F_AX5xErrMsg:= 'F168 =  Process data mapping: MDT - Memory problem';
	16#F169: F_AX5xErrMsg:= 'F169 =  Process data mapping: Internal error';
	16#F16A: F_AX5xErrMsg:= 'F16A =  Process data mapping: MDT - Too many IDN"s';
	16#F16B: F_AX5xErrMsg:= 'F16B =  Process data mapping: AT-list,  double listed entry found';
	16#F16C: F_AX5xErrMsg:= 'F16C =  Process data mapping: MDT-list,  double listed entry found';
	16#F180: F_AX5xErrMsg:= 'F180 =  Internal communication: SCI - Control card to front card';
	16#F183: F_AX5xErrMsg:= 'F183 =  Feedback (general): Commutation feedback is not feedback 1';
	16#F184: F_AX5xErrMsg:= 'F184 =  Feedback "general": Commutation feedback is not feedback 2';
	16#F185: F_AX5xErrMsg:= 'F185 =  Internal communication: SCI - Control card to front card';
	16#F186: F_AX5xErrMsg:= 'F186 =  Internal communication: SCI - Control card to front card';
	16#F187: F_AX5xErrMsg:= 'F187 =  Internal communication: SCI - Control card to front card';
	16#F188: F_AX5xErrMsg:= 'F188 =  Internal communication: SCI - Control card to front card';
	16#F189: F_AX5xErrMsg:= 'F189 =  Internal communication: SCI - Control card to front card';
	16#F18A: F_AX5xErrMsg:= 'F18A =  Internal communication: SCI - Control card to front card';
	16#F18B: F_AX5xErrMsg:= 'F18B =  Internal communication: SCI - Control card to front card';
	16#F18C: F_AX5xErrMsg:= 'F18C =  Internal communication: SCI - Front card to control card';
	16#F18D: F_AX5xErrMsg:= 'F18D =  Internal communication: SCI - Front card to control card';
	16#F18E: F_AX5xErrMsg:= 'F18E =  Internal communication: SCI - Front card to control card';
	16#F18F: F_AX5xErrMsg:= 'F18F =  Internal communication: SCI - Front card to control card';
	16#F190: F_AX5xErrMsg:= 'F190 =  Internal communication: SPI - Control card to front card';
	16#F191: F_AX5xErrMsg:= 'F191 =  Internal communication: SPI - Control card to front card';
	16#F192: F_AX5xErrMsg:= 'F192 =  Internal communication: SPI - Control card to front card';
	16#F193: F_AX5xErrMsg:= 'F193 =  Internal communication: SPI - Control card to front card';
	16#F194: F_AX5xErrMsg:= 'F194 =  Internal communication: SPI - Front card to Control card';
	16#F195: F_AX5xErrMsg:= 'F195 =  Internal communication: SPI - Front card to Control card';
	16#F196: F_AX5xErrMsg:= 'F196 =  Internal communication: SPI - Front card to Control card';
	16#F197: F_AX5xErrMsg:= 'F197 =  Internal communication: SPI - Front card to Control card';
	16#F198: F_AX5xErrMsg:= 'F198 =  Internal communication: SPI - Control card to front card';
	16#F199: F_AX5xErrMsg:= 'F199 =  Internal communication: SPI - Control card to front card';
	16#F19A: F_AX5xErrMsg:= 'F19A =  Internal communication: SPI - Control card to front card';
	16#F19B: F_AX5xErrMsg:= 'F19B =  Internal communication: SPI - Control card to front card';
	16#F19C: F_AX5xErrMsg:= 'F19C =  Internal communication: SPI - Control card to front card';
	16#F19D: F_AX5xErrMsg:= 'F19D =  Internal communication: SPI - Control card to front card';
	16#F19E: F_AX5xErrMsg:= 'F19E =  Internal communication: SPI - Control card to front card';
	16#F1A0: F_AX5xErrMsg:= 'F1A0 =  Internal communication: SCI - Control card to front card';
	16#F1A1: F_AX5xErrMsg:= 'F1A1 =  Internal communication: SCI - Control card to front card';
	16#F1B0: F_AX5xErrMsg:= 'F1B0 =  Communication Control - Option pcb: Init failed.';
	16#F1B1: F_AX5xErrMsg:= 'F1B1 =  Option slot card: Commutation feedback not supported.';
	16#F1B2: F_AX5xErrMsg:= 'F1B2 =  Option slot card: Additional feedback not feedback 2.';
	16#F1B5: F_AX5xErrMsg:= 'F1B5 =  Internal communication: SCI - Control card to option card';
	16#F1B6: F_AX5xErrMsg:= 'F1B6 =  Internal communication: SCI - Control card to option card';
	16#F1B7: F_AX5xErrMsg:= 'F1B7 =  Internal communication: SCI - Control card to option card';
	16#F1B8: F_AX5xErrMsg:= 'F1B8 =  Internal communication: SCI - Control card to option card';
	16#F1B9: F_AX5xErrMsg:= 'F1B9 =  Internal communication: SCI - Control card to option card';
	16#F1BA: F_AX5xErrMsg:= 'F1BA =  Internal communication: SCI - Control card to option card';
	16#F1BB: F_AX5xErrMsg:= 'F1BB =  Internal communication: SCI - Control card to option card';
	16#F1BC: F_AX5xErrMsg:= 'F1BC =  Internal communication: SPI - Control card to option card';
	16#F1BD: F_AX5xErrMsg:= 'F1BD =  Internal communication: SPI - Control card to option card';
	16#F1D0: F_AX5xErrMsg:= 'F1D0 =  Internal communication: SCI - Control card to option card';
	16#F1D1: F_AX5xErrMsg:= 'F1D1 =  Internal communication: The feedback unit don"t supports the requested action.';
	16#F290: F_AX5xErrMsg:= 'F290 =  Cycle time out: High prioritise processes';
	16#F291: F_AX5xErrMsg:= 'F291 =  Time out: Low prioritise processes';
	16#F292: F_AX5xErrMsg:= 'F292 =  Internal task scheduler error';
	16#F2A0: F_AX5xErrMsg:= 'F2A0 =  Commutation error';
	16#F2A1: F_AX5xErrMsg:= 'F2A1 =  Overcurrent error motor, measuring limit reached (X13 / X23).';
	16#F2A2: F_AX5xErrMsg:= 'F2A2 =  Processing unit periphery: Initialisation failed';
	16#F2A3: F_AX5xErrMsg:= 'F2A3 =  Current controler: Internal use failed';
	16#F2A4: F_AX5xErrMsg:= 'F2A4 =  Internal error';
	16#F2A5: F_AX5xErrMsg:= 'F2A5 =  Internal error';
	16#F2A7: F_AX5xErrMsg:= 'F2A7 =  Torque off triggered from "shorted coils brake" or "DC brake"';
	16#F2E1: F_AX5xErrMsg:= 'F2E1 =  Velocity Control: Control deviation monitoring failed';
	16#F320: F_AX5xErrMsg:= 'F320 =  Discontinuity in the position command value';
	16#F321: F_AX5xErrMsg:= 'F321 =  Excessive position deviation';
	16#F323: F_AX5xErrMsg:= 'F323 =  Parameter error';
	16#F324: F_AX5xErrMsg:= 'F324 =  Excessive position command value deviation.';
	16#F325: F_AX5xErrMsg:= 'F325 =  Following distance calculation limit exceeded.';
	16#F326: F_AX5xErrMsg:= 'F326 =  Additional position deviation monitoring';
	16#F330: F_AX5xErrMsg:= 'F330 =  Position control - Interpolator error';
	16#F331: F_AX5xErrMsg:= 'F331 =  Position control - Interpolator error';
	16#F332: F_AX5xErrMsg:= 'F332 =  Position control - Interpolator error';
	16#F333: F_AX5xErrMsg:= 'F333 =  Position control - Interpolator error';
	16#F340: F_AX5xErrMsg:= 'F340 =  Position offset invalid';
	16#F341: F_AX5xErrMsg:= 'F341 =  Position offset: No position offset excisting';
	16#F342: F_AX5xErrMsg:= 'F342 =  Position offset: Offset can"t be activated. Modulo calculation is active.';
	16#F343: F_AX5xErrMsg:= 'F343 =  Position offset: No position offset excisting';
	16#F344: F_AX5xErrMsg:= 'F344 =  Position offset: The position offset change is greater than the modulo value.';
	16#F350: F_AX5xErrMsg:= 'F350 =  Modulo Calculation: No saved data could be loaded.';
	16#F351: F_AX5xErrMsg:= 'F351 =  Modulo Calculation: Initialization data invalid.';
	16#F352: F_AX5xErrMsg:= 'F352 =  Modulo Calculation: No saved data available.';
	16#F353: F_AX5xErrMsg:= 'F353 =  Modulo Calculation: Saving of the initialization data failed.';
	16#F354: F_AX5xErrMsg:= 'F354 =  Modulo Calculation: Saving of the modulo data failed.';
	16#F355: F_AX5xErrMsg:= 'F355 =  Modulo Calculation: The absolute range of encoder 1 is too small.';
	16#F356: F_AX5xErrMsg:= 'F356 =  Modulo Calculation: The absolute range of encoder 2 is too small.';
	16#F357: F_AX5xErrMsg:= 'F357 =  Modulo Calculation: Init failed because the feedback position is invalid.';
	16#F360: F_AX5xErrMsg:= 'F360 =  Initialisation of the device: failed';
	16#F361: F_AX5xErrMsg:= 'F361 =  Initialisation of the device: failed';
	16#F362: F_AX5xErrMsg:= 'F362 =  Initialisation of the device: Failed - Firmware checksum';
	16#F363: F_AX5xErrMsg:= 'F363 =  Initialisation of the device: Failed - Firmware checksum';
	16#F3A0: F_AX5xErrMsg:= 'F3A0 =  Device initialisation: Invalid state';
	16#F3A1: F_AX5xErrMsg:= 'F3A1 =  Device initialisation: Invalid state';
	16#F3A3: F_AX5xErrMsg:= 'F3A3 =  Start of the device front unit failed';
	16#F3A4: F_AX5xErrMsg:= 'F3A4 =  Device initialisation: Option card - Feedback DSP failed';
	16#F3A5: F_AX5xErrMsg:= 'F3A5 =  Device initialisation: Option card - FPGA test failed';
	16#F3A6: F_AX5xErrMsg:= 'F3A6 =  Device initialisation: Serial flash,  firmware info not readable';
	16#F3A7: F_AX5xErrMsg:= 'F3A7 =  Device initialisation: Serial flash,  boot loader info not readable';
	16#F3A8: F_AX5xErrMsg:= 'F3A8 =  Device initialisation: Serial flash,  directory not readable';
	16#F3A9: F_AX5xErrMsg:= 'F3A9 =  Explicit Device Identification: Read of the data failed.';
	16#F3AA: F_AX5xErrMsg:= 'F3AA =  Explicit Device Identification: Write of the data failed.';
	16#F3AB: F_AX5xErrMsg:= 'F3AB =  Explicit Device Identification: Write of the data failed.';
	16#F3C0: F_AX5xErrMsg:= 'F3C0 =  Error management: Invalid value in P-0-0350';
	16#F3C1: F_AX5xErrMsg:= 'F3C1 =  Error management: Internal error';
	16#F3C2: F_AX5xErrMsg:= 'F3C2 =  Error management: Command error';
	16#F3C3: F_AX5xErrMsg:= 'F3C3 =  Error management: Command error';
	16#F3C4: F_AX5xErrMsg:= 'F3C4 =  Error management: Init failed';
	16#F3C5: F_AX5xErrMsg:= 'F3C5 =  Error management: Got no timer';
	16#F3D0: F_AX5xErrMsg:= 'F3D0 =  Propagated error received,  react with "Torque off".';
	16#F3D1: F_AX5xErrMsg:= 'F3D1 =  Propagated error received,  react with "Shorted coils brake".';
	16#F3D2: F_AX5xErrMsg:= 'F3D2 =  Propagated error received, react with "Open loop ramp".';
	16#F3D3: F_AX5xErrMsg:= 'F3D3 =  Propagated error received,  react with "Closed loop ramp".';
	16#F3D4: F_AX5xErrMsg:= 'F3D4 =  Propagated error received,  react with "Gantry brake".';
	16#F401: F_AX5xErrMsg:= 'F401 =  EtherCAT slave controller: Internal test failed';
	16#F402: F_AX5xErrMsg:= 'F402 =  EtherCAT slave controller: Syncmanager - start adress';
	16#F403: F_AX5xErrMsg:= 'F403 =  EtherCAT slave controller: Syncmanager - adress range';
	16#F404: F_AX5xErrMsg:= 'F404 =  EtherCAT slave controller: Syncmanager - size';
	16#F405: F_AX5xErrMsg:= 'F405 =  EtherCAT slave controller: Syncmanager - parameter';
	16#F406: F_AX5xErrMsg:= 'F406 =  EtherCAT slave controller: Syncmanager - internal error';
	16#F407: F_AX5xErrMsg:= 'F407 =  EtherCAT slave controller (MDT): Syncmanager - parameter';
	16#F408: F_AX5xErrMsg:= 'F408 =  EtherCAT slave controller (AT): Syncmanager - parameter';
	16#F409: F_AX5xErrMsg:= 'F409 =  Distributed clocks: Sync0 - Cycle time';
	16#F410: F_AX5xErrMsg:= 'F410 =  Distributed clocks: Sync0 - Not enabled';
	16#F411: F_AX5xErrMsg:= 'F411 =  Distributed clocks: Sync0 - Impulse length';
	16#F412: F_AX5xErrMsg:= 'F412 =  Distributed clocks: Sync1 - Cycle time';
	16#F413: F_AX5xErrMsg:= 'F413 =  Distributed clocks: Sync1 - Not enabled';
	16#F414: F_AX5xErrMsg:= 'F414 =  Distributed clocks: hardware sync';
	16#F415: F_AX5xErrMsg:= 'F415 =  Distributed clocks: Process data synchronization lost';
	16#F420: F_AX5xErrMsg:= 'F420 =  EtherCAT slave controller: Invalid port configuration';
	16#F440: F_AX5xErrMsg:= 'F440 =  Dynamic SyncManager: IO-Cylce counter error';
	16#F441: F_AX5xErrMsg:= 'F441 =  Dynamic SyncManager: Required SyncManager not enabled.';
	16#F4A0: F_AX5xErrMsg:= 'F4A0 =  SoE Communication: Reset command failed';
	16#F4A1: F_AX5xErrMsg:= 'F4A1 =  SoE Communication: Internal error';
	16#F4A2: F_AX5xErrMsg:= 'F4A2 =  SoE Communication: Internal error';
	16#F4A3: F_AX5xErrMsg:= 'F4A3 =  SoE Communication: Internal error';
	16#F4A4: F_AX5xErrMsg:= 'F4A4 =  SoE Communication: Internal error';
	16#F4A5: F_AX5xErrMsg:= 'F4A5 =  SoE Communication: Parameter error';
	16#F4A6: F_AX5xErrMsg:= 'F4A6 =  SoE Communication: Drive notification failed';
	16#F4A7: F_AX5xErrMsg:= 'F4A7 =  SoE Communication: Internal error';
	16#F4A8: F_AX5xErrMsg:= 'F4A8 =  SoE Communication: Internal error';
	16#F4A9: F_AX5xErrMsg:= 'F4A9 =  SoE Communication: Internal error';
	16#F4AA: F_AX5xErrMsg:= 'F4AA =  SoE Communication: Internal error';
	16#F4AB: F_AX5xErrMsg:= 'F4AB =  SoE Communication: Parameter error';
	16#F500: F_AX5xErrMsg:= 'F500 =  Internal error.';
	16#F503: F_AX5xErrMsg:= 'F503 =  Internal communication error';
	16#F504: F_AX5xErrMsg:= 'F504 =  A/D converter: Reference voltage invalid';
	16#F505: F_AX5xErrMsg:= 'F505 =  Firmware: Analysis of the A/D-Converter defective';
	16#F506: F_AX5xErrMsg:= 'F506 =  Internal communication error';
	16#F508: F_AX5xErrMsg:= 'F508 =  Firmware: Unknown nominal current.';
	16#F50A: F_AX5xErrMsg:= 'F50A =  A/D-Converter: DC-Link - measuring error';
	16#F50B: F_AX5xErrMsg:= 'F50B =  A/D-Converter: DC-Link - measuring error';
	16#F50C: F_AX5xErrMsg:= 'F50C =  A/D-Converter: DC-Link - Measuring error';
	16#F50D: F_AX5xErrMsg:= 'F50D =  A/D-Converter: DC-Link - Measuring error';
	16#F50E: F_AX5xErrMsg:= 'F50E =  A/D-Converter: Measuring error - Umains';
	16#F50F: F_AX5xErrMsg:= 'F50F =  A/D-Converter: Measuring error - Modul temperature';
	16#F510: F_AX5xErrMsg:= 'F510 =  A/D-Converter: Not ready to enable';
	16#F511: F_AX5xErrMsg:= 'F511 =  Voltage calibration failed';
	16#F580: F_AX5xErrMsg:= 'F580 =  External Periphery - Control card: Internal error';
	16#F581: F_AX5xErrMsg:= 'F581 =  External Periphery - Control card: Reading the ESC-eeprom failed';
	16#F582: F_AX5xErrMsg:= 'F582 =  External Periphery - Control card: Writing the ESC-eeprom failed';
	16#F583: F_AX5xErrMsg:= 'F583 =  External Periphery - Control card: Reading the ESC-eeprom failed';
	16#F584: F_AX5xErrMsg:= 'F584 =  External Periphery - Control card: Reading the ESC-eeprom failed';
	16#F585: F_AX5xErrMsg:= 'F585 =  External Periphery - Control card: Reading the ESC-eeprom failed';
	16#F586: F_AX5xErrMsg:= 'F586 =  External Periphery - Control card: Checking the ESC-eeprom failed';
	16#F587: F_AX5xErrMsg:= 'F587 =  External Periphery - Control card: Checking the ESC-eeprom failed';
	16#F588: F_AX5xErrMsg:= 'F588 =  External Periphery: SPI - Timeout';
	16#F589: F_AX5xErrMsg:= 'F589 =  External Periphery - Control card: Reading the ESC-eeprom failed';
	16#F58A: F_AX5xErrMsg:= 'F58A =  External Periphery - Control card: Writing the ESC-eeprom failed';
	16#F58B: F_AX5xErrMsg:= 'F58B =  External Periphery - Control card: Writing the ESC-eeprom failed';
	16#F58C: F_AX5xErrMsg:= 'F58C =  External Periphery - Control card: Writing the ESC-eeprom failed';
	16#F58D: F_AX5xErrMsg:= 'F58D =  External Periphery - Control card: Writing the ESC-eeprom failed';
	16#F590: F_AX5xErrMsg:= 'F590 =  External Periphery - Control card: ADC - Initialisation failed';
	16#F591: F_AX5xErrMsg:= 'F591 =  External Periphery - Initialisation failed';
	16#F600: F_AX5xErrMsg:= 'F600 =  Calibrate commutation offset error.';
	16#F601: F_AX5xErrMsg:= 'F601 =  Calibrate commutation offset error.';
	16#F602: F_AX5xErrMsg:= 'F602 =  Calibrate commutation offset error.';
	16#F603: F_AX5xErrMsg:= 'F603 =  Calibrate commutation offset error.';
	16#F604: F_AX5xErrMsg:= 'F604 =  Current calibration error.';
	16#F605: F_AX5xErrMsg:= 'F605 =  Current calibration error.';
	16#F606: F_AX5xErrMsg:= 'F606 =  Current calibration error.';
	16#F607: F_AX5xErrMsg:= 'F607 =  Current calibration error.';
	16#F608: F_AX5xErrMsg:= 'F608 =  Current calibration error.';
	16#F609: F_AX5xErrMsg:= 'F609 =  Current calibration error.';
	16#F60A: F_AX5xErrMsg:= 'F60A =  Current calibration error.';
	16#F60B: F_AX5xErrMsg:= 'F60B =  Current calibration error.';
	16#F60C: F_AX5xErrMsg:= 'F60C =  Current calibration error.';
	16#F60D: F_AX5xErrMsg:= 'F60D =  Calibrate commutation offset error.';
	16#F60E: F_AX5xErrMsg:= 'F60E =  Calibrate commutation offset error.';
	16#F610: F_AX5xErrMsg:= 'F610 =  Current calibration error.';
	16#F611: F_AX5xErrMsg:= 'F611 =  Current calibration error.';
	16#F612: F_AX5xErrMsg:= 'F612 =  Current calibration error.';
	16#F700: F_AX5xErrMsg:= 'F700 =  Feedback "general": Initialization';
	16#F701: F_AX5xErrMsg:= 'F701 =  Feedback "general": Initialization - parameter channel';
	16#F702: F_AX5xErrMsg:= 'F702 =  Feedback "1": Position invalid.';
	16#F703: F_AX5xErrMsg:= 'F703 =  Feedback "general": Feedback error';
	16#F704: F_AX5xErrMsg:= 'F704 =  Feedback "general": Over voltage - supply voltage';
	16#F705: F_AX5xErrMsg:= 'F705 =  Feedback "general": Under voltage - Supply voltage';
	16#F706: F_AX5xErrMsg:= 'F706 =  Feedback "general": Internal error.';
	16#F707: F_AX5xErrMsg:= 'F707 =  Feedback "general": Lost feedback';
	16#F708: F_AX5xErrMsg:= 'F708 =  Feedback "general": Found different feedback in the digital name plate.';
	16#F709: F_AX5xErrMsg:= 'F709 =  Feedback "2": Position invalid.';
	16#F70A: F_AX5xErrMsg:= 'F70A =  Feedback "1": Error.';
	16#F70B: F_AX5xErrMsg:= 'F70B =  Feedback "2": error.';
	16#F70E: F_AX5xErrMsg:= 'F70E =  Feedback "1": error.';
	16#F70F: F_AX5xErrMsg:= 'F70F =  Feedback "2": error';
	16#F712: F_AX5xErrMsg:= 'F712 =  Feedback "general": Power settings';
	16#F713: F_AX5xErrMsg:= 'F713 =  Feedback "general": process data channel settings';
	16#F714: F_AX5xErrMsg:= 'F714 =  Feedback "general": parameter channel settings';
	16#F715: F_AX5xErrMsg:= 'F715 =  Internal communication: SPI - Front card to Option card';
	16#F716: F_AX5xErrMsg:= 'F716 =  Internal communication: SPI - Front card to Option card';
	16#F717: F_AX5xErrMsg:= 'F717 =  Feedback "general": Initialisation failed';
	16#F718: F_AX5xErrMsg:= 'F718 =  Feedback "1": Data invalid (SPI Error).';
	16#F719: F_AX5xErrMsg:= 'F719 =  Option card, Feedback "1": error';
	16#F71A: F_AX5xErrMsg:= 'F71A =  Option card, Feedback "2": error';
	16#F720: F_AX5xErrMsg:= 'F720 =  Feedback "general": Initialisation failed';
	16#F721: F_AX5xErrMsg:= 'F721 =  Feedback "general": Initialisation failed';
	16#F722: F_AX5xErrMsg:= 'F722 =  Feedback "general": Initialisation failed';
	16#F723: F_AX5xErrMsg:= 'F723 =  Feedback "general": Initialisation failed';
	16#F724: F_AX5xErrMsg:= 'F724 =  Feedback "general": Initialisation failed';
	16#F725: F_AX5xErrMsg:= 'F725 =  Feedback "general": Initialisation failed';
	16#F726: F_AX5xErrMsg:= 'F726 =  Feedback "general": Save digital name plate failed.';
	16#F727: F_AX5xErrMsg:= 'F727 =  Feedback "general" Save position offset failed.';
	16#F728: F_AX5xErrMsg:= 'F728 =  Feedback "general": Position initialisation failed.';
	16#F729: F_AX5xErrMsg:= 'F729 =  Feedback "general": Scan feedback failed.';
	16#F72A: F_AX5xErrMsg:= 'F72A =  Feedback "general": Internal error';
	16#F72B: F_AX5xErrMsg:= 'F72B =  Feedback "general": Internal error';
	16#F72C: F_AX5xErrMsg:= 'F72C =  Feedback "general": Internal error';
	16#F72E: F_AX5xErrMsg:= 'F72E =  Feedback "general": Internal error';
	16#F72F: F_AX5xErrMsg:= 'F72F =  Feedback "general": Internal error';
	16#F730: F_AX5xErrMsg:= 'F730 =  Feedback "general": Internal error';
	16#F731: F_AX5xErrMsg:= 'F731 =  Feedback "general": Initialisation failed';
	16#F732: F_AX5xErrMsg:= 'F732 =  Feedback "general": Save digital name plate failed.';
	16#F733: F_AX5xErrMsg:= 'F733 =  Feedback "general" Save position offset failed.';
	16#F734: F_AX5xErrMsg:= 'F734 =  Feedback "general": Position initialisation failed.';
	16#F735: F_AX5xErrMsg:= 'F735 =  Feedback "general": Position initialisation failed.';
	16#F736: F_AX5xErrMsg:= 'F736 =  Feedback "general": Data transfer failed.';
	16#F737: F_AX5xErrMsg:= 'F737 =  Feedback "general": Data transfer failed.';
	16#F738: F_AX5xErrMsg:= 'F738 =  Feedback "general": Data transfer failed.';
	16#F739: F_AX5xErrMsg:= 'F739 =  Feedback "general": Wrong feedback';
	16#F73A: F_AX5xErrMsg:= 'F73A =  Feedback "general": Resolution has been incorrectly parameterised';
	16#F73B: F_AX5xErrMsg:= 'F73B =  Feedback "general": Resolution has been incorrectly parameterised';
	16#F73C: F_AX5xErrMsg:= 'F73C =  Feedback "general": Resolution per rotation has been incorrectly parameterised';
	16#F73D: F_AX5xErrMsg:= 'F73D =  Feedback "general": Length of the signal period has been incorrectly parameterised';
	16#F73E: F_AX5xErrMsg:= 'F73E =  Feedback "general": Data transfer failed.';
	16#F73F: F_AX5xErrMsg:= 'F73F =  Feedback "general": Feedback id has been incorrectly parameterised';
	16#F740: F_AX5xErrMsg:= 'F740 =  Feedback "general": Initialisation failed';
	16#F741: F_AX5xErrMsg:= 'F741 =  Feedback "general": Unknown multiturn position';
	16#F742: F_AX5xErrMsg:= 'F742 =  Feedback "general": Invalid commutation offset';
	16#F743: F_AX5xErrMsg:= 'F743 =  Feeback"general": No feedback connector choosen';
	16#F744: F_AX5xErrMsg:= 'F744 =  Feeback"general": Wrong feedback connector choosen';
	16#F745: F_AX5xErrMsg:= 'F745 =  Feedback "general": Data transfer failed.';
	16#F747: F_AX5xErrMsg:= 'F747 =  Feedback "general": Parameter invalid.';
	16#F748: F_AX5xErrMsg:= 'F748 =  Feeback"general": Parameter channel - Position invalid';
	16#F749: F_AX5xErrMsg:= 'F749 =  Feedback "general": Parameter invalid.';
	16#F74A: F_AX5xErrMsg:= 'F74A =  Feedback "general": Parameter invalid';
	16#F74B: F_AX5xErrMsg:= 'F74B =  Feedback "general": Save data failed';
	16#F74C: F_AX5xErrMsg:= 'F74C =  Feedback "general": Save data failed';
	16#F74D: F_AX5xErrMsg:= 'F74D =  Feedback "general": Parameter invalid';
	16#F74E: F_AX5xErrMsg:= 'F74E =  Feedback "general": Parameter invalid';
	16#F770: F_AX5xErrMsg:= 'F770 =  Feedback SSI: Invalid parameter.';
	16#F771: F_AX5xErrMsg:= 'F771 =  Feedback SSI: Single turn resolution to high.';
	16#F772: F_AX5xErrMsg:= 'F772 =  Feedback SSI: Mulit turn resolution to high.';
	16#F780: F_AX5xErrMsg:= 'F780 =  Feedback "general": Data transfer failed.';
	16#F781: F_AX5xErrMsg:= 'F781 =  Feedback "general": Data transfer failed.';
	16#F782: F_AX5xErrMsg:= 'F782 =  Feedback "general": Initialisation failed';
	16#F783: F_AX5xErrMsg:= 'F783 =  Feedback "general": Initialisation failed';
	16#F784: F_AX5xErrMsg:= 'F784 =  Feedback "general": Initialisation failed';
	16#F785: F_AX5xErrMsg:= 'F785 =  Feedback "general": Initialisation failed';
	16#F786: F_AX5xErrMsg:= 'F786 =  Feedback "general": Initialisation failed';
	16#F787: F_AX5xErrMsg:= 'F787 =  Feedback "general": Initialisation failed';
	16#F788: F_AX5xErrMsg:= 'F788 =  Feedback "general": Encoder error';
	16#F789: F_AX5xErrMsg:= 'F789 =  Feedback "general": Initialisation failed';
	16#F78A: F_AX5xErrMsg:= 'F78A =  Feedback "general": Initialisation failed';
	16#F78B: F_AX5xErrMsg:= 'F78B =  Feedback "general": Initialisation failed';
	16#F78C: F_AX5xErrMsg:= 'F78C =  Feedback "general": Initialisation failed';
	16#F78D: F_AX5xErrMsg:= 'F78D =  Feedback "general": Initialisation failed';
	16#F78E: F_AX5xErrMsg:= 'F78E =  Feedback "general": Initialisation failed';
	16#F78F: F_AX5xErrMsg:= 'F78F =  Feedback "general": Initialisation failed';
	16#F791: F_AX5xErrMsg:= 'F791 =  Feedback parameter channel error (Endat).';
	16#F792: F_AX5xErrMsg:= 'F792 =  Feedback parameter channel error (Endat).';
	16#F793: F_AX5xErrMsg:= 'F793 =  Feedback parameter channel error (Endat).';
	16#F794: F_AX5xErrMsg:= 'F794 =  Endat: Feedback scan invalid.';
	16#F7C0: F_AX5xErrMsg:= 'F7C0 =  Feedback parameter channel error (Biss).';
	16#F7C1: F_AX5xErrMsg:= 'F7C1 =  Feedback parameter channel error (Biss).';
	16#F7C2: F_AX5xErrMsg:= 'F7C2 =  Feedback parameter channel error (Biss).';
	16#F7C3: F_AX5xErrMsg:= 'F7C3 =  Feedback parameter channel init error (Biss).';
	16#F7C4: F_AX5xErrMsg:= 'F7C4 =  Feedback parameter channel error (Biss).';
	16#F7C5: F_AX5xErrMsg:= 'F7C5 =  Feedback parameter channel init error (Biss).';
	16#F7C6: F_AX5xErrMsg:= 'F7C6 =  Feedback parameter channel init error (Biss).';
	16#F7C7: F_AX5xErrMsg:= 'F7C7 =  Feedback parameter channel init error (Biss).';
	16#F7C8: F_AX5xErrMsg:= 'F7C8 =  Feedback parameter channel init error (Biss).';
	16#F7C9: F_AX5xErrMsg:= 'F7C9 =  Feedback parameter channel init error (Biss).';
	16#F7CA: F_AX5xErrMsg:= 'F7CA =  Feedback parameter channel init error (Biss).';
	16#F7CB: F_AX5xErrMsg:= 'F7CB =  Feedback parameter channel init error (Biss).';
	16#F7CC: F_AX5xErrMsg:= 'F7CC =  Feedback parameter channel init error (Biss).';
	16#F7CD: F_AX5xErrMsg:= 'F7CD =  Feedback parameter channel error (Biss).';
	16#F7CE: F_AX5xErrMsg:= 'F7CE =  Feedback parameter channel error (Biss).';
	16#F7CF: F_AX5xErrMsg:= 'F7CF =  Biss: Feedback scan invalid.';
	16#F7D0: F_AX5xErrMsg:= 'F7D0 =  Feedback parameter channel error (Biss).';
	16#F7D1: F_AX5xErrMsg:= 'F7D1 =  Feedback parameter channel error (Biss).';
	16#F7D2: F_AX5xErrMsg:= 'F7D2 =  Feedback parameter channel error (Biss).';
	16#F7D3: F_AX5xErrMsg:= 'F7D3 =  Feedback parameter channel error (Biss).';
	16#F7D4: F_AX5xErrMsg:= 'F7D4 =  Feedback parameter channel error (Biss).';
	16#F7D5: F_AX5xErrMsg:= 'F7D5 =  Feedback parameter channel error (Biss).';
	16#F7D6: F_AX5xErrMsg:= 'F7D6 =  Feedback parameter channel error (Biss).';
	16#F7D7: F_AX5xErrMsg:= 'F7D7 =  Feedback parameter channel error (Biss).';
	16#F7D8: F_AX5xErrMsg:= 'F7D8 =  Feedback parameter channel error (Biss).';
	16#F800: F_AX5xErrMsg:= 'F800 =  Feedback parameter channel init error (Hiperface): by read manufacturer parameter';
	16#F801: F_AX5xErrMsg:= 'F801 =  Feedback parameter channel init error (Hiperface): by read feedback status';
	16#F802: F_AX5xErrMsg:= 'F802 =  Feedback ôHiperfaceö init error - Parameter channel';
	16#F803: F_AX5xErrMsg:= 'F803 =  Feedback parameter channel init error (Hiperface): unknown name plate';
	16#F804: F_AX5xErrMsg:= 'F804 =  Feedback parameter channel init error (Hiperface): singleturn resolution over 32bit';
	16#F805: F_AX5xErrMsg:= 'F805 =  Feedback parameter channel init error (Hiperface): multiturn resolution over 12 bit';
	16#F806: F_AX5xErrMsg:= 'F806 =  Feedback parameter channel init error (Hiperface): not enough memory';
	16#F807: F_AX5xErrMsg:= 'F807 =  Feedback parameter channel init error (Hiperface): "scan feedback" not valid for this command';
	16#F808: F_AX5xErrMsg:= 'F808 =  Feedback parameter channel init error (Hiperface): open internal interface';
	16#F809: F_AX5xErrMsg:= 'F809 =  Feedback parameter channel init error (Hiperface): internal unknown state';
	16#F80A: F_AX5xErrMsg:= 'F80A =  Feedback parameter channel error (Hiperface): feedback denied command';
	16#F80B: F_AX5xErrMsg:= 'F80B =  Feedback parameter channel init error (Hiperface): feedback denied reset command';
	16#F80C: F_AX5xErrMsg:= 'F80C =  Feedback parameter channel error (Hiperface): unable to clear datafields';
	16#F80D: F_AX5xErrMsg:= 'F80D =  Feedback parameter channel error (Hiperface): sci frame error';
	16#F80E: F_AX5xErrMsg:= 'F80E =  Feedback parameter channel init error (Hiperface): sci parity error';
	16#F80F: F_AX5xErrMsg:= 'F80F =  Feedback parameter channel init error (Hiperface): wrong checksum';
	16#F810: F_AX5xErrMsg:= 'F810 =  Feedback parameter channel init error (Hiperface): wrong address';
	16#F811: F_AX5xErrMsg:= 'F811 =  Feedback ôHiperfaceö init error . parameter channel';
	16#F812: F_AX5xErrMsg:= 'F812 =  Feedback parameter channel init error (Hiperface): wrong response';
	16#F813: F_AX5xErrMsg:= 'F813 =  Feedback parameter channel init error (Hiperface): sci error';
	16#F840: F_AX5xErrMsg:= 'F840 =  Feedback analog comutaion channel init error.';
	16#F841: F_AX5xErrMsg:= 'F841 =  Feedback analog comutaion channel init error.';
	16#F842: F_AX5xErrMsg:= 'F842 =  Feedback analog comutaion channel init error.';
	16#F843: F_AX5xErrMsg:= 'F843 =  Feedback analog comutation channel init error.';
	16#F844: F_AX5xErrMsg:= 'F844 =  Error, feedback parameter channel, can"t create object.';
	16#F845: F_AX5xErrMsg:= 'F845 =  Feedback analog init error.';
	16#F846: F_AX5xErrMsg:= 'F846 =  Feedback analog commutation part error.';
	16#F850: F_AX5xErrMsg:= 'F850 =  One cable feedback: Link missing';
	16#F851: F_AX5xErrMsg:= 'F851 =  One cable feedback: Initialization failed';
	16#F852: F_AX5xErrMsg:= 'F852 =  One cable feedback: Position error limit exceeded';
	16#F853: F_AX5xErrMsg:= 'F853 =  One cable feedback: Get position - Timeout';
	16#F854: F_AX5xErrMsg:= 'F854 =  One cable feedback: Out of memory';
	16#F855: F_AX5xErrMsg:= 'F855 =  One cable feedback: Parameter error';
	16#F856: F_AX5xErrMsg:= 'F856 =  One cable feedback: Write config failed';
	16#F857: F_AX5xErrMsg:= 'F857 =  One cable feedback: Read of the cyclic data failed';
	16#F858: F_AX5xErrMsg:= 'F858 =  One cable feedback: Internal error';
	16#F859: F_AX5xErrMsg:= 'F859 =  One cable feedback: Write system control failed';
